M_StartMoveBoxToRoundBelt_ClampB := TRUE; // Method end
END_METHOD

(* This method is used to setting the Fanuc Robot Action " Pickup box from PulloutConveyor , only clampA"
*)
METHOD M_StartPullOutConveyorPickUpBox_ClampA : BOOL
VAR_INPUT
	ClampA_Address : E_PullOutConveyorPosition;
	BoxReady : BOOL; // True : Pullout conveyor box is ready. accroding ClampA target slide is ready or not.
END_VAR
VAR_INST
	_Area : ST_IntToBool;
    _Address_ClampA : ST_IntToBool;
END_VAR
// Set target area is round belt
_Area.nInt := E_RobotArea.PullOutConveyor;
// Select pullout conveyor slide
IF ClampA_Address = E_PullOutConveyorPosition.I3_Slide THEN
	_Address_ClampA.nInt := 1;
ELSIF ClampA_Address = E_PullOutConveyorPosition.I4_Slide THEN
	_Address_ClampA.nInt := 2;
ELSE
	// Wrong command, return
	RETURN ;
END_IF
// Send robot target area data
_DO3.nArea1 := _Area.BitList.Bit0;
_DO3.nArea2 := _Area.BitList.Bit1;
_DO3.nArea3 := _Area.BitList.Bit2;
_DO3.nArea4 := _Area.BitList.Bit3;

// Send robot target address data
_DO3.nAddress1 := _Address_ClampA.BitList.Bit0;
_DO3.nAddress2 := _Address_ClampA.BitList.Bit1;
_DO3.nAddress3 := _Address_ClampA.BitList.Bit2;
_DO3.nAddress4 := _Address_ClampA.BitList.Bit3;
_DO3.nAddress5 := _Address_ClampA.BitList.Bit4;
_DO3.nAddress6 := _Address_ClampA.BitList.Bit5;
_DO3.nAddress7 := _Address_ClampA.BitList.Bit6;

_DO3.bGet := TRUE; // Pickup action
_DO3.bExecute := TRUE;

_DO3.bContinue := BoxReady;

M_StartPullOutConveyorPickUpBox_ClampA := true; // Method end
END_METHOD

(* This method is used to setting the Fanuc Robot Action " Pickup box from PulloutConveyor , only clampB"
*)
METHOD M_StartPullOutConveyorPickUpBox_ClampB : BOOL
VAR_INPUT
	ClampB_Address :E_PullOutConveyorPosition;
	BoxReady : BOOL; // True : Pullout conveyor box is ready. accroding ClampA target slide is ready or not.
END_VAR
VAR_INST
	_Area : ST_IntToBool;
    _Address_ClampB : ST_IntToBool;
END_VAR
// Set target area is round belt
_Area.nInt := E_RobotArea.PullOutConveyor;
// Select pullout conveyor slide
IF ClampB_Address = E_PullOutConveyorPosition.I3_Slide THEN
	_Address_ClampB.nInt := 1;
ELSIF ClampB_Address = E_PullOutConveyorPosition.I4_Slide THEN
	_Address_ClampB.nInt := 2;
ELSE
	// Wrong command, return
	RETURN ;
END_IF

// Send robot target area data
_DO4.nArea1 := _Area.BitList.Bit0;
_DO4.nArea2 := _Area.BitList.Bit1;
_DO4.nArea3 := _Area.BitList.Bit2;
_DO4.nArea4 := _Area.BitList.Bit3;

// Send robot target address data
_DO4.nAddress1 := _Address_ClampB.BitList.Bit0;
_DO4.nAddress2 := _Address_ClampB.BitList.Bit1;
_DO4.nAddress3 := _Address_ClampB.BitList.Bit2;
_DO4.nAddress4 := _Address_ClampB.BitList.Bit3;
_DO4.nAddress5 := _Address_ClampB.BitList.Bit4;
_DO4.nAddress6 := _Address_ClampB.BitList.Bit5;
_DO4.nAddress7 := _Address_ClampB.BitList.Bit6;

_DO4.bGet := TRUE; // Pickup action
_DO4.bExecute := TRUE;

_DO4.bContinue := BoxReady;

M_StartPullOutConveyorPickUpBox_ClampB := true; // Method end
END_METHOD

(* This method is used to setting the Fanuc Robot Action " Pickup box from PulloutConveyor, both clamp"
*)
METHOD M_StartPullOutConveyorPickUpBox_ClampBoth : BOOL
VAR_INPUT
	ClampA_Address : E_PullOutConveyorPosition;
	ClampB_Address : E_PullOutConveyorPosition;
	BoxReady_1 : BOOL; // TRUE : 1st target slide box is ready
	BoxReady_2 : BOOL; // True : 2nd target slide box is ready
END_VAR
VAR_INST
	_Area : ST_IntToBool;
    _Address_ClampA : ST_IntToBool;
    _Address_ClampB : ST_IntToBool;
END_VAR
// Set target area is round belt
_Area.nInt := E_RobotArea.PullOutConveyor;

// Select ClampA target address
IF ClampA_Address = E_PullOutConveyorPosition.I3_Slide THEN
    _Address_ClampA.nInt := 1;
ELSIF ClampA_Address = E_PullOutConveyorPosition.I4_Slide THEN
    _Address_ClampA.nInt := 2;
ELSE
    // Wrong command, return
    RETURN;
END_IF

// Select ClampB target address
IF ClampB_Address = E_PullOutConveyorPosition.I3_Slide THEN
    _Address_ClampB.nInt := 1;
ELSIF ClampB_Address = E_PullOutConveyorPosition.I4_Slide THEN
    _Address_ClampB.nInt := 2;
ELSE
    // Wrong command, return
    RETURN;
END_IF

// Send robot target area data
_DO3.nArea1 := _Area.BitList.Bit0;
_DO3.nArea2 := _Area.BitList.Bit1;
_DO3.nArea3 := _Area.BitList.Bit2;
_DO3.nArea4 := _Area.BitList.Bit3;

_DO4.nArea1 := _Area.BitList.Bit0;
_DO4.nArea2 := _Area.BitList.Bit1;
_DO4.nArea3 := _Area.BitList.Bit2;
_DO4.nArea4 := _Area.BitList.Bit3;

// Send robot target address data
_DO3.nAddress1 := _Address_ClampA.BitList.Bit0;
_DO3.nAddress2 := _Address_ClampA.BitList.Bit1;
_DO3.nAddress3 := _Address_ClampA.BitList.Bit2;
_DO3.nAddress4 := _Address_ClampA.BitList.Bit3;
_DO3.nAddress5 := _Address_ClampA.BitList.Bit4;
_DO3.nAddress6 := _Address_ClampA.BitList.Bit5;
_DO3.nAddress7 := _Address_ClampA.BitList.Bit6;

_DO4.nAddress1 := _Address_ClampB.BitList.Bit0;
_DO4.nAddress2 := _Address_ClampB.BitList.Bit1;
_DO4.nAddress3 := _Address_ClampB.BitList.Bit2;
_DO4.nAddress4 := _Address_ClampB.BitList.Bit3;
_DO4.nAddress5 := _Address_ClampB.BitList.Bit4;
_DO4.nAddress6 := _Address_ClampB.BitList.Bit5;
_DO4.nAddress7 := _Address_ClampB.BitList.Bit6;

_DO3.bGet := TRUE;
_DO4.bGet := TRUE;

_DO3.bExecute := TRUE;
_DO4.bExecute := TRUE;

_DO3.bContinue := BoxReady_1;
_DO4.bContinue := BoxReady_2;

M_StartPullOutConveyorPickUpBox_ClampBoth := true; // Method end
END_METHOD

METHOD PUBLIC M_StartRobotAbsMove : BOOL
VAR_INPUT
	GetBox		: BOOL;
	UseClampA	: BOOL;
	UseClampB   : BOOL;
	Area : E_RobotArea;
	
	
	ClampA_Address	: INT;
	ClampB_Address	: INT;

	BoxReady_1 : BOOL;
	BoxReady_2 : BOOL;
	
END_VAR

VAR_INST
	_Area	: ST_IntToBool;
	_Address_ClampA : ST_IntToBool;
    _Address_ClampB : ST_IntToBool;
END_VAR
//Set target area
_Area.nInt :=Area;

IF UseClampA THEN
	_Address_ClampA.nInt:=ClampA_Address;
	_DO3.nArea1 := _Area.BitList.Bit0;
	_DO3.nArea2 := _Area.BitList.Bit1;
	_DO3.nArea3 := _Area.BitList.Bit2;
	_DO3.nArea4 := _Area.BitList.Bit3;

	_DO3.nAddress1 := _Address_ClampA.BitList.Bit0;
	_DO3.nAddress2 := _Address_ClampA.BitList.Bit1;
	_DO3.nAddress3 := _Address_ClampA.BitList.Bit2;
	_DO3.nAddress4 := _Address_ClampA.BitList.Bit3;
	_DO3.nAddress5 := _Address_ClampA.BitList.Bit4;
	_DO3.nAddress6 := _Address_ClampA.BitList.Bit5;
	_DO3.nAddress7 := _Address_ClampA.BitList.Bit6;
	_DO3.bGet := GetBox;
	_DO3.bExecute := TRUE;
	_DO3.bContinue := BoxReady_1;	
END_IF

IF UseClampB THEN
	_Address_ClampB.nInt:=ClampB_Address;
	_DO4.nArea1 := _Area.BitList.Bit0;
	_DO4.nArea2 := _Area.BitList.Bit1;
	_DO4.nArea3 := _Area.BitList.Bit2;
	_DO4.nArea4 := _Area.BitList.Bit3;
	
	_DO4.nAddress1 := _Address_ClampB.BitList.Bit0;
	_DO4.nAddress2 := _Address_ClampB.BitList.Bit1;
	_DO4.nAddress3 := _Address_ClampB.BitList.Bit2;
	_DO4.nAddress4 := _Address_ClampB.BitList.Bit3;
	_DO4.nAddress5 := _Address_ClampB.BitList.Bit4;
	_DO4.nAddress6 := _Address_ClampB.BitList.Bit5;
	_DO4.nAddress7 := _Address_ClampB.BitList.Bit6;
	_DO4.bGet := GetBox;
	_DO4.bExecute := TRUE;
	_DO4.bContinue := BoxReady_2;	
END_IF

M_StartRobotAbsMove :=TRUE;




















M_StartRobotAbsMove:=TRUE;
END_METHOD

METHOD M_StartWarehouseMoveAction_ClampA : BOOL
VAR_INPUT
	WareHouseSelect : E_WareHouse;
	Info : ST_WareHouseCoordinates; // Input Warehouse with robot move parameter for pickup box;
	ClampAction :E_ClampAction;
	BoxReady : BOOL;
END_VAR
VAR_OUTPUT
	Error : BOOL;
	ErrMsg :T_MaxString;
END_VAR
VAR_INST
	_Layer : ST_IntToBool;
	_Slide : ST_IntToBool;
END_VAR
// Set target warehouse
CASE WareHouseSelect OF
    E_WareHouse.WareHouseA:
        _DO1.bTargetWareHouseA := TRUE;
        _DO1.bTargetWareHouseB := FALSE;
    E_WareHouse.WareHouseB:
        _DO1.bTargetWareHouseA := FALSE;
        _DO1.bTargetWareHouseB := TRUE;
ELSE
    _DO1.bTargetWareHouseA := FALSE;
    _DO1.bTargetWareHouseB := FALSE;
    Error                  := TRUE;
    ErrMsg                 := 'ClampA target warehouse out of range';
	RETURN;
END_CASE

// Set Warehouse coordinates
_Layer.nInt := info.Layer;
_Slide.nInt := info.Slide;

// Send Layer data to robot
_DO1.nLayer1 := _Layer.BitList.Bit0;
_DO1.nLayer2 := _Layer.BitList.Bit1;
_DO1.nLayer3 := _Layer.BitList.Bit2;
_DO1.nLayer4 := _Layer.BitList.Bit3;

// Send Slide data to Robot
_DO1.nSlide1 := _Slide.BitList.Bit0;
_DO1.nSlide2 := _Slide.BitList.Bit1;
_DO1.nSlide3 := _Slide.BitList.Bit2;
_DO1.nSlide4 := _Slide.BitList.Bit3;
_DO1.nSlide5 := _Slide.BitList.Bit4;

// Send clamp action to robot
CASE ClampAction OF
	E_ClampAction.PickUp:
		_DO1.bGet := TRUE;
	E_ClampAction.Place:
		_DO1.bGet := FALSE;
ELSE
	Error := TRUE;
	ErrMsg := 'Clamp action not defined';
	RETURN;
END_CASE

// Send action data to robot
_DO1.bExecute := NOT Error;
_DO1.bContinue := BoxReady;
M_StartWarehouseMoveAction_ClampA := NOT Error; // Method end
END_METHOD

METHOD M_StartWarehouseMoveAction_ClampB : BOOL
VAR_INPUT
	WareHouseSelect : E_WareHouse;
	Info : ST_WareHouseCoordinates; // Input Warehouse with robot move parameter for pickup box;
	ClampAction :E_ClampAction;
	BoxReady : BOOL;
END_VAR
VAR_OUTPUT
	Error : BOOL;
	ErrMsg :T_MaxString;
END_VAR
VAR_INST
	_Layer : ST_IntToBool;
	_Slide : ST_IntToBool;
END_VAR
// Set target warehouse
CASE WareHouseSelect OF
    E_WareHouse.WareHouseA:
        _DO2.bTargetWareHouseA := TRUE;
        _DO2.bTargetWareHouseB := FALSE;
    E_WareHouse.WareHouseB:
        _DO2.bTargetWareHouseA := FALSE;
        _DO2.bTargetWareHouseB := TRUE;
ELSE
    _DO2.bTargetWareHouseA := FALSE;
    _DO2.bTargetWareHouseB := FALSE;
    Error                  := TRUE;
    ErrMsg                 := 'ClampB target warehouse out of range';
	RETURN;
END_CASE

// Set Warehouse coordinates
_Layer.nInt := info.Layer;
_Slide.nInt := info.Slide;

// Send Layer data to robot
_DO2.nLayer1 := _Layer.BitList.Bit0;
_DO2.nLayer2 := _Layer.BitList.Bit1;
_DO2.nLayer3 := _Layer.BitList.Bit2;
_DO2.nLayer4 := _Layer.BitList.Bit3;

// Send Slide data to Robot
_DO2.nSlide1 := _Slide.BitList.Bit0;
_DO2.nSlide2 := _Slide.BitList.Bit1;
_DO2.nSlide3 := _Slide.BitList.Bit2;
_DO2.nSlide4 := _Slide.BitList.Bit3;
_DO2.nSlide5 := _Slide.BitList.Bit4;

// Send clamp action to robot
CASE ClampAction OF
	E_ClampAction.PickUp:
		_DO2.bGet := TRUE;
	E_ClampAction.Place:
		_DO2.bGet := FALSE;
ELSE
	Error := TRUE;
	ErrMsg := 'Clamp action not defined';
	RETURN;
END_CASE

// Send action data to robot
_DO2.bExecute := NOT Error;
_DO2.bContinue := BoxReady;

M_StartWarehouseMoveAction_ClampB := NOT Error; // Method End
END_METHOD

METHOD M_StartWarehouseMoveAction_ClampBoth : BOOL
VAR_INPUT
	WareHouseSelect : E_WareHouse;
	ClampA_Info : ST_WareHouseCoordinates; // Input Warehouse with robot move parameter for pickup box;
	ClampB_Info : ST_WareHouseCoordinates; // Input Warehouse with robot move parameter for pickup box;
	ClampAction_A : E_ClampAction;
	ClampAction_B : E_ClampAction;
	BoxReady_1st : BOOL; // Box is arrived, ready to pickup
	BoxReady_2nd : BOOL; // Box is arrived, ready to pickup
END_VAR
VAR_OUTPUT
	Error : BOOL;
	ErrMsg :T_MaxString;
END_VAR
VAR_INST
	_LayerClampA :ST_IntToBool;
	_SlideClampA : ST_IntToBool;
	_LayerClampB : ST_IntToBool;
	_SLideClampB : ST_IntToBool;
END_VAR
// Set target warehouse
CASE WareHouseSelect OF
    E_WareHouse.WareHouseA:
        _DO1.bTargetWareHouseA := TRUE;
        _DO1.bTargetWareHouseB := FALSE;
        _DO2.bTargetWareHouseA := TRUE;
        _DO2.bTargetWareHouseB := FALSE;
    E_WareHouse.WareHouseB:
        _DO1.bTargetWareHouseA := FALSE;
        _DO1.bTargetWareHouseB := TRUE;
        _DO2.bTargetWareHouseA := FALSE;
        _DO2.bTargetWareHouseB := TRUE;
ELSE
    _DO1.bTargetWareHouseA := FALSE;
    _DO1.bTargetWareHouseB := FALSE;
    _DO2.bTargetWareHouseA := FALSE;
    _DO2.bTargetWareHouseB := FALSE;
    Error                  := TRUE;
    ErrMsg                 := 'Clamp target warehouse out of range';
    RETURN;
END_CASE

// Assign coordinates 
_LayerClampA.nInt := ClampA_Info.Layer;
_SlideClampA.nInt := ClampA_Info.Slide;
_LayerClampB.nInt := ClampB_Info.Layer;
_SlideClampB.nInt := ClampB_Info.Slide;

// Send Layer data to Robot
_DO1.nLayer1 := _LayerClampA.BitList.Bit0;
_DO1.nLayer2 := _LayerClampA.BitList.Bit1;
_DO1.nLayer3 := _LayerClampA.BitList.Bit2;
_DO1.nLayer4 := _LayerClampA.BitList.Bit3;
_DO2.nLayer1 := _LayerClampB.BitList.Bit0;
_DO2.nLayer2 := _LayerClampB.BitList.Bit1;
_DO2.nLayer3 := _LayerClampB.BitList.Bit2;
_DO2.nLayer4 := _LayerClampB.BitList.Bit3;
// Send Slide data to Robot
_DO1.nSlide1 := _SlideClampA.BitList.Bit0;
_DO1.nSlide2 := _SlideClampA.BitList.Bit1;
_DO1.nSlide3 := _SlideClampA.BitList.Bit2;
_DO1.nSlide4 := _SlideClampA.BitList.Bit3;
_DO1.nSlide5 := _SlideClampA.BitList.Bit4;

_DO2.nSlide1 := _SlideClampB.BitList.Bit0;
_DO2.nSlide2 := _SlideClampB.BitList.Bit1;
_DO2.nSlide3 := _SlideClampB.BitList.Bit2;
_DO2.nSlide4 := _SlideClampB.BitList.Bit3;
_DO2.nSlide5 := _SlideClampB.BitList.Bit4;

// Set clamp action 
CASE ClampAction_A OF
	E_ClampAction.PickUp:
		_DO1.bGet := TRUE;
	E_ClampAction.Place:
		_DO1.bGet := FALSE;
ELSE
	Error := TRUE;
	ErrMsg := 'ClampA action not defined';
	RETURN;
END_CASE

// Set clamp action
CASE ClampAction_B OF
	E_ClampAction.PickUp:
		_DO2.bGet := TRUE;
	E_ClampAction.Place:
		_DO2.bGet := FALSE;
ELSE
	Error := TRUE;
	ErrMsg := 'ClampB action not defined';
	RETURN;	
END_CASE

// set execute
_DO1.bExecute := NOT Error;
_DO2.bExecute := NOT Error;

_DO1.bContinue := BoxReady_1st;
_DO2.bContinue := BoxReady_2nd;

M_StartWarehouseMoveAction_ClampBoth := NOT Error; // Method end
END_METHOD

METHOD M_StartWareHousePickUpBox_ClampA : Bool
VAR_INPUT
	WareHouseSelect : E_WareHouse;
	Info : ST_WareHouseCoordinates; // Input Warehouse with robot move parameter for pickup box;
	BoxReady_1st : BOOL;
END_VAR
VAR_INST
	_Layer : ST_IntToBool;
	_Slide : ST_IntToBool;
END_VAR
// Send target warehouse to robot
IF WareHouseSelect = E_WareHouse.WareHouseA THEN
	_DO1.bTargetWareHouseA := TRUE;
	_DO1.bTargetWareHouseB := FALSE;
ELSIF WareHouseSelect = E_WareHouse.WareHouseB THEN
	_DO1.bTargetWareHouseA := FALSE;
	_DO1.bTargetWareHouseB := TRUE;
ELSE
	_DO1.bTargetWareHouseA := FALSE;
	_DO1.bTargetWareHouseB := FALSE;
END_IF

// Assign coordinates 
_Layer.nInt := info.Layer;
_Slide.nInt := info.Slide;

// Send Layer data to Robot
_DO1.nLayer1 := _Layer.BitList.Bit0;
_DO1.nLayer2 := _Layer.BitList.Bit1;
_DO1.nLayer3 := _Layer.BitList.Bit2;
_DO1.nLayer4 := _Layer.BitList.Bit3;

// Send Slide data to Robot
_DO1.nSlide1 := _Slide.BitList.Bit0;
_DO1.nSlide2 := _Slide.BitList.Bit1;
_DO1.nSlide3 := _Slide.BitList.Bit2;
_DO1.nSlide4 := _Slide.BitList.Bit3;
_DO1.nSlide5 := _Slide.BitList.Bit4;

// Send action data to robot
_DO1.bGet := TRUE; // PickUp
// Send execute command 
_DO1.bExecute := TRUE;
_DO1.bContinue := BoxReady_1st;
M_StartWareHousePickUpBox_ClampA := TRUE; // Method end
END_METHOD

METHOD M_StartWareHousePickUpBox_ClampB : BOOL
VAR_INPUT
	WareHouseSelect : E_WareHouse;
	Info : ST_WareHouseCoordinates; // Input Warehouse with robot move parameter for pickup box;
	BoxReady_2nd : BOOL;
END_VAR
VAR_INST
	_Layer : ST_IntToBool;
	_Slide : ST_IntToBool;
END_VAR
// Send target warehouse to robot
IF WareHouseSelect = E_WareHouse.WareHouseA THEN
    _DO2.bTargetWareHouseA := TRUE;
    _DO2.bTargetWareHouseB := FALSE;
ELSIF WareHouseSelect = E_WareHouse.WareHouseB THEN
    _DO2.bTargetWareHouseA := FALSE;
    _DO2.bTargetWareHouseB := TRUE;
ELSE
    _DO2.bTargetWareHouseA := FALSE;
    _DO2.bTargetWareHouseB := FALSE;
END_IF

// Assign coordinates 
_Layer.nInt := info.Layer;
_Slide.nInt := info.Slide;

// Send Layer data to Robot
_DO2.nLayer1 := _Layer.BitList.Bit0;
_DO2.nLayer2 := _Layer.BitList.Bit1;
_DO2.nLayer3 := _Layer.BitList.Bit2;
_DO2.nLayer4 := _Layer.BitList.Bit3;

// Send Slide data to Robot
_DO2.nSlide1 := _Slide.BitList.Bit0;
_DO2.nSlide2 := _Slide.BitList.Bit1;
_DO2.nSlide3 := _Slide.BitList.Bit2;
_DO2.nSlide4 := _Slide.BitList.Bit3;
_DO2.nSlide5 := _Slide.BitList.Bit4;

// Send action data to robot
_DO2.bGet := TRUE; // PickUp
// Send execute command 
_DO2.bExecute := TRUE;
_DO2.bContinue:=BoxReady_2nd;
M_StartWareHousePickUpBox_ClampB := TRUE; // Method end
END_METHOD

METHOD M_StartWareHousePickUpBox_ClampBoth : BOOL
VAR_INPUT
	WareHouseSelect : E_WareHouse;
	ClampA_Info : ST_WareHouseCoordinates; // Input Warehouse with robot move parameter for pickup box;
	ClampB_Info : ST_WareHouseCoordinates; // Input Warehouse with robot move parameter for pickup box;
	BoxReady_1st : BOOL; // Box is arrived, ready to pickup
	BoxReady_2nd : BOOL; // Box is arrived, ready to pickup
END_VAR
VAR_OUTPUT
	Error : BOOL;
	ErrMsg :T_MaxString;
END_VAR
VAR_INST
	_LayerClampA : ST_IntToBool;
	_SlideClampA : ST_IntToBool;
	_LayerClampB : ST_IntToBool;
	_SlideClampB : ST_IntToBool;
END_VAR
// Set target warehouse
CASE WareHouseSelect OF
    E_WareHouse.WareHouseA:
        _DO1.bTargetWareHouseA := TRUE;
        _DO1.bTargetWareHouseB := FALSE;
        _DO2.bTargetWareHouseA := TRUE;
        _DO2.bTargetWareHouseB := FALSE;
    E_WareHouse.WareHouseB:
        _DO1.bTargetWareHouseA := FALSE;
        _DO1.bTargetWareHouseB := TRUE;
        _DO2.bTargetWareHouseA := FALSE;
        _DO2.bTargetWareHouseB := TRUE;
ELSE
    _DO1.bTargetWareHouseA := FALSE;
    _DO1.bTargetWareHouseB := FALSE;
    _DO2.bTargetWareHouseA := FALSE;
    _DO2.bTargetWareHouseB := FALSE;
    Error                  := TRUE;
    ErrMsg                 := 'Clamp target warehouse out of range';
    RETURN;
END_CASE

// Assign coordinates 
_LayerClampA.nInt := ClampA_Info.Layer;
_SlideClampA.nInt := ClampA_Info.Slide;
_LayerClampB.nInt := ClampB_Info.Layer;
_SlideClampB.nInt := ClampB_Info.Slide;

// Send Layer data to Robot
_DO1.nLayer1 := _LayerClampA.BitList.Bit0;
_DO1.nLayer2 := _LayerClampA.BitList.Bit1;
_DO1.nLayer3 := _LayerClampA.BitList.Bit2;
_DO1.nLayer4 := _LayerClampA.BitList.Bit3;

_DO2.nLayer1 := _LayerClampB.BitList.Bit0;
_DO2.nLayer2 := _LayerClampB.BitList.Bit1;
_DO2.nLayer3 := _LayerClampB.BitList.Bit2;
_DO2.nLayer4 := _LayerClampB.BitList.Bit3;
// Send Slide data to Robot
_DO1.nSlide1 := _SlideClampA.BitList.Bit0;
_DO1.nSlide2 := _SlideClampA.BitList.Bit1;
_DO1.nSlide3 := _SlideClampA.BitList.Bit2;
_DO1.nSlide4 := _SlideClampA.BitList.Bit3;
_DO1.nSlide5 := _SlideClampA.BitList.Bit4;

_DO2.nSlide1 := _SlideClampB.BitList.Bit0;
_DO2.nSlide2 := _SlideClampB.BitList.Bit1;
_DO2.nSlide3 := _SlideClampB.BitList.Bit2;
_DO2.nSlide4 := _SlideClampB.BitList.Bit3;
_DO2.nSlide5 := _SlideClampB.BitList.Bit4;

// Send action data to robot
_DO1.bGet := TRUE; // ClampA PickUp
_DO2.bGet := TRUE; // ClampB PickUp
// Send execute command 
_DO1.bExecute := NOT Error;
_DO2.bExecute := NOT Error;

_DO1.bContinue := BoxReady_1st;
_DO2.bContinue := BoxReady_2nd;

M_StartWareHousePickUpBox_ClampBoth := NOT Error; // Method end
END_METHOD

METHOD M_StartWareHousePlaceBox_ClampA : Bool
VAR_INPUT
	WareHouseSelect : E_WareHouse;
	Info : ST_WareHouseCoordinates; // Input Warehouse with robot move parameter for pickup box;
	BoxReady_1st : BOOL;
END_VAR
VAR_INST
	_Layer : ST_IntToBool;
	_Slide : ST_IntToBool;
END_VAR
// Send target warehouse to robot
IF WareHouseSelect = E_WareHouse.WareHouseA THEN
	_DO1.bTargetWareHouseA := TRUE;
	_DO1.bTargetWareHouseB := FALSE;
ELSIF WareHouseSelect = E_WareHouse.WareHouseB THEN
	_DO1.bTargetWareHouseA := FALSE;
	_DO1.bTargetWareHouseB := TRUE;
ELSE
	_DO1.bTargetWareHouseA := FALSE;
	_DO1.bTargetWareHouseB := FALSE;
END_IF

// Assign coordinates 
_Layer.nInt := info.Layer;
_Slide.nInt := info.Slide;

// Send Layer data to Robot
_DO1.nLayer1 := _Layer.BitList.Bit0;
_DO1.nLayer2 := _Layer.BitList.Bit1;
_DO1.nLayer3 := _Layer.BitList.Bit2;
_DO1.nLayer4 := _Layer.BitList.Bit3;

// Send Slide data to Robot
_DO1.nSlide1 := _Slide.BitList.Bit0;
_DO1.nSlide2 := _Slide.BitList.Bit1;
_DO1.nSlide3 := _Slide.BitList.Bit2;
_DO1.nSlide4 := _Slide.BitList.Bit3;
_DO1.nSlide5 := _Slide.BitList.Bit4;

// Send action data to robot
_DO1.bGet := FALSE; // PickUp
// Send execute command 
_DO1.bExecute := TRUE;
_DO1.bContinue := BoxReady_1st;
M_StartWareHousePlaceBox_ClampA := TRUE; // Method end
END_METHOD

METHOD M_StartWareHousePlaceBox_ClampB : BOOL
VAR_INPUT
	WareHouseSelect : E_WareHouse;
	Info : ST_WareHouseCoordinates; // Input Warehouse with robot move parameter for pickup box;
	BoxReady_2nd : BOOL;
END_VAR
VAR_INST
	_Layer : ST_IntToBool;
	_Slide : ST_IntToBool;
END_VAR
// Send target warehouse to robot
IF WareHouseSelect = E_WareHouse.WareHouseA THEN
    _DO2.bTargetWareHouseA := TRUE;
    _DO2.bTargetWareHouseB := FALSE;
ELSIF WareHouseSelect = E_WareHouse.WareHouseB THEN
    _DO2.bTargetWareHouseA := FALSE;
    _DO2.bTargetWareHouseB := TRUE;
ELSE
    _DO2.bTargetWareHouseA := FALSE;
    _DO2.bTargetWareHouseB := FALSE;
END_IF

// Assign coordinates 
_Layer.nInt := info.Layer;
_Slide.nInt := info.Slide;

// Send Layer data to Robot
_DO2.nLayer1 := _Layer.BitList.Bit0;
_DO2.nLayer2 := _Layer.BitList.Bit1;
_DO2.nLayer3 := _Layer.BitList.Bit2;
_DO2.nLayer4 := _Layer.BitList.Bit3;

// Send Slide data to Robot
_DO2.nSlide1 := _Slide.BitList.Bit0;
_DO2.nSlide2 := _Slide.BitList.Bit1;
_DO2.nSlide3 := _Slide.BitList.Bit2;
_DO2.nSlide4 := _Slide.BitList.Bit3;
_DO2.nSlide5 := _Slide.BitList.Bit4;

// Send action data to robot
_DO2.bGet := FALSE; // PickUp
// Send execute command 
_DO2.bExecute := TRUE;
_DO2.bContinue:=BoxReady_2nd;
M_StartWareHousePlaceBox_ClampB := TRUE; // Method end
END_METHOD

METHOD M_StartWareHousePlaceUpBox_ClampBoth : BOOL
VAR_INPUT
	WareHouseSelect : E_WareHouse;
	ClampA_Info : ST_WareHouseCoordinates; // Input Warehouse with robot move parameter for pickup box;
	ClampB_Info : ST_WareHouseCoordinates; // Input Warehouse with robot move parameter for pickup box;
	BoxReady_1st : BOOL; // Box is arrived, ready to pickup
	BoxReady_2nd : BOOL; // Box is arrived, ready to pickup
END_VAR
VAR_OUTPUT
	Error : BOOL;
	ErrMsg :T_MaxString;
END_VAR
VAR_INST
	_LayerClampA : ST_IntToBool;
	_SlideClampA : ST_IntToBool;
	_LayerClampB : ST_IntToBool;
	_SlideClampB : ST_IntToBool;
END_VAR
// Set target warehouse
CASE WareHouseSelect OF
    E_WareHouse.WareHouseA:
        _DO1.bTargetWareHouseA := TRUE;
        _DO1.bTargetWareHouseB := FALSE;
        _DO2.bTargetWareHouseA := TRUE;
        _DO2.bTargetWareHouseB := FALSE;
    E_WareHouse.WareHouseB:
        _DO1.bTargetWareHouseA := FALSE;
        _DO1.bTargetWareHouseB := TRUE;
        _DO2.bTargetWareHouseA := FALSE;
        _DO2.bTargetWareHouseB := TRUE;
ELSE
    _DO1.bTargetWareHouseA := FALSE;
    _DO1.bTargetWareHouseB := FALSE;
    _DO2.bTargetWareHouseA := FALSE;
    _DO2.bTargetWareHouseB := FALSE;
    Error                  := TRUE;
    ErrMsg                 := 'Clamp target warehouse out of range';
    RETURN;
END_CASE

// Assign coordinates 
_LayerClampA.nInt := ClampA_Info.Layer;
_SlideClampA.nInt := ClampA_Info.Slide;
_LayerClampB.nInt := ClampB_Info.Layer;
_SlideClampB.nInt := ClampB_Info.Slide;

// Send Layer data to Robot
_DO1.nLayer1 := _LayerClampA.BitList.Bit0;
_DO1.nLayer2 := _LayerClampA.BitList.Bit1;
_DO1.nLayer3 := _LayerClampA.BitList.Bit2;
_DO1.nLayer4 := _LayerClampA.BitList.Bit3;

_DO2.nLayer1 := _LayerClampB.BitList.Bit0;
_DO2.nLayer2 := _LayerClampB.BitList.Bit1;
_DO2.nLayer3 := _LayerClampB.BitList.Bit2;
_DO2.nLayer4 := _LayerClampB.BitList.Bit3;
// Send Slide data to Robot
_DO1.nSlide1 := _SlideClampA.BitList.Bit0;
_DO1.nSlide2 := _SlideClampA.BitList.Bit1;
_DO1.nSlide3 := _SlideClampA.BitList.Bit2;
_DO1.nSlide4 := _SlideClampA.BitList.Bit3;
_DO1.nSlide5 := _SlideClampA.BitList.Bit4;

_DO2.nSlide1 := _SlideClampB.BitList.Bit0;
_DO2.nSlide2 := _SlideClampB.BitList.Bit1;
_DO2.nSlide3 := _SlideClampB.BitList.Bit2;
_DO2.nSlide4 := _SlideClampB.BitList.Bit3;
_DO2.nSlide5 := _SlideClampB.BitList.Bit4;

// Send action data to robot
_DO1.bGet := FALSE; // ClampA PickUp
_DO2.bGet := FALSE; // ClampB PickUp
// Send execute command 
_DO1.bExecute := NOT Error;
_DO2.bExecute := NOT Error;

_DO1.bContinue := BoxReady_1st;
_DO2.bContinue := BoxReady_2nd;

M_StartWareHousePlaceUpBox_ClampBoth := NOT Error; // Method end
END_METHOD

METHOD M_SwitchRSR3 : BOOL
VAR_INPUT
END_VAR
END_METHOD

PROPERTY Read_OffsetP : INT
GET
Read_OffsetP := _DI6;
END_GET
END_PROPERTY

PROPERTY Read_OffsetR : INT
GET
Read_OffsetR := _DI7;
END_GET
END_PROPERTY

PROPERTY Read_OffsetW : INT
GET
Read_OffsetW := _DI5;
END_GET
END_PROPERTY

PROPERTY Read_OffsetX : INT
GET
Read_OffsetX := _DI2;
END_GET
END_PROPERTY

PROPERTY Read_OffsetY : INT
GET
Read_OffsetY := _DI3;
END_GET
END_PROPERTY

PROPERTY Read_OffsetZ : INT
GET
Read_OffsetZ := _DI4;
END_GET
END_PROPERTY

PROPERTY ReadDataCommand : BOOL;
SET
_DO6.ReadPara_Execute := BOOL_TO_BIT(ReadDataCommand);
END_SET
END_PROPERTY

PROPERTY ReadWrite_Address : Int
SET
_Do14 := ReadWrite_Address;
END_SET
END_PROPERTY

PROPERTY ReadWrite_Area : E_RobotArea
SET
_Do13 := ReadWrite_Area;
END_SET
END_PROPERTY

(* This variable is used to define read/write offset data clamp A
*)
PROPERTY ReadWrite_ClampA : BOOL
SET
_DO6.ClampA :=  BOOL_TO_BIT(ReadWrite_ClampA );
END_SET
END_PROPERTY

(* This variable is used to define read/write offset data clamp B
*)
PROPERTY ReadWrite_ClampB : BOOL
SET
_DO6.ClampB :=BOOL_TO_BIT( ReadWrite_ClampB);
END_SET
END_PROPERTY

(* This variable is used to define read/write offset data warehouse A
*)
PROPERTY ReadWrite_WareHouseA : BOOL
SET
_DO6.WareHouseA := BOOL_TO_BIT(ReadWrite_WareHouseA);
END_SET
END_PROPERTY

(* This variable is used to define read/write offset data warehouse B
*)
PROPERTY ReadWrite_WareHouseB : BOOL
SET
_DO6.WarehouseB := BOOL_TO_BIT(ReadWrite_WareHouseB);
END_SET
END_PROPERTY

(*Fanuc robot ready to work for command (Warehouse、AbsMove)*)
PROPERTY ReadyOperation : Bool
GET
ReadyOperation := _RSR1_Ready;
END_GET
END_PROPERTY

PROPERTY ReadySetParameter : Bool
GET
ReadySetParameter := _RSR3_Ready;
END_GET
END_PROPERTY

METHOD ReBoot
VAR_INPUT
END_VAR
eState := E_MethodStatus_Basic.STATE_DORMANT;
END_METHOD

PROPERTY SlideIndex : INT
SET
_DO16 := SlideIndex;
END_SET
END_PROPERTY

PROPERTY Status : ST_FanucUI1
GET
Status := _UI1;
END_GET
END_PROPERTY

METHOD Update : BOOL
VAR_INPUT
END_VAR
// Robot -> PLC 4 byte 外圍設備Output(Fanuc Robot的外圍)
MEMMOVE(
destAddr:=ADR(_UO1)
,srcAddr:=ADR(_rawIn_UI[0])
,n:=4
);

// PLC -> Robot 外圍設備Input(Fanuc Robot的外圍)
MEMMOVE(
destAddr:=ADR(_rawOut_UO[0])
,srcAddr:=ADR(_UI1)
,n:=4
);
// PLC -> Robot Digital Output 2byte(send the command to Fanuc Robot), Warehouse Robot move ClampA
MEMMOVE(
destAddr:=ADR(_rawOut_DO[0])
,srcAddr:=ADR(_DO1)
,n:=2 
);
// PLC -> Robot Digital Output 2byte(send the command to Fanuc Robot), Warehouse Robot move ClampB
MEMMOVE(
destAddr:=ADR(_rawOut_DO[2])
,srcAddr:=ADR(_DO2)
,n:=2 
);
// PLC -> Robot Digital Output 2byte(send the command to Fanuc Robot), ABS Robot move ClampA
MEMMOVE(
destAddr:=ADR(_rawOut_DO[4])
,srcAddr:=ADR(_DO3)
,n:=2 
);
// PLC -> Robot Digital Output 2byte(send the command to Fanuc Robot), ABS Robot move ClampA
MEMMOVE(
destAddr:=ADR(_rawOut_DO[6])
,srcAddr:=ADR(_DO4)
,n:=2 
);
// PLC -> Robot Digital output 2byte(send the command to Fanuc Robot), General Command
MEMMOVE(
destAddr:=ADR(_rawOut_DO[8])
,srcAddr:=ADR(_DO5)
,n:=2 
);
MEMMOVE(
destAddr:=ADR(_rawOut_DO[10])
,srcAddr:=ADR(_DO6)
,n:=2 
);
MEMMOVE(
destAddr:=ADR(_rawOut_DO[12])
,srcAddr:=ADR(_DO7)
,n:=2 
);
MEMMOVE(
destAddr:=ADR(_rawOut_DO[14])
,srcAddr:=ADR(_DO8)
,n:=2 
);
MEMMOVE(
destAddr:=ADR(_rawOut_DO[16])
,srcAddr:=ADR(_DO9)
,n:=2 
);

MEMMOVE(
destAddr:=ADR(_rawOut_DO[18])
,srcAddr:=ADR(_DO10)
,n:=2 
);
MEMMOVE(
destAddr:=ADR(_rawOut_DO[20])
,srcAddr:=ADR(_DO11)
,n:=2 
);
MEMMOVE(
destAddr:=ADR(_rawOut_DO[22])
,srcAddr:=ADR(_DO12)
,n:=2 
);
MEMMOVE(
destAddr:=ADR(_rawOut_DO[24])
,srcAddr:=ADR(_DO13)
,n:=2 
);
MEMMOVE(
destAddr:=ADR(_rawOut_DO[26])
,srcAddr:=ADR(_DO14)
,n:=2 
);
MEMMOVE(
destAddr:=ADR(_rawOut_DO[28])
,srcAddr:=ADR(_DO15)
,n:=2 
);
MEMMOVE(
destAddr:=ADR(_rawOut_DO[30])
,srcAddr:=ADR(_DO16)
,n:=2 
);


// Robot -> PLC Digital Input 3byte(Send Robot Status to PLC), All service
MEMMOVE(
destAddr:=ADR(_DI1)
,srcAddr:=ADR(_rawIn_DI[0])
,n:=3
);

MEMMOVE(
destAddr:=ADR(_DI2)
,srcAddr:=ADR(_rawIn_DI[3])
,n:=2
);
MEMMOVE(
destAddr:=ADR(_DI3)
,srcAddr:=ADR(_rawIn_DI[5])
,n:=2
);
MEMMOVE(
destAddr:=ADR(_DI4)
,srcAddr:=ADR(_rawIn_DI[7])
,n:=2
);
MEMMOVE(
destAddr:=ADR(_DI5)
,srcAddr:=ADR(_rawIn_DI[9])
,n:=2
);
MEMMOVE(
destAddr:=ADR(_DI6)
,srcAddr:=ADR(_rawIn_DI[11])
,n:=2
);
MEMMOVE(
destAddr:=ADR(_DI7)
,srcAddr:=ADR(_rawIn_DI[13])
,n:=2
);
MEMMOVE(
destAddr:=ADR(_DI8)
,srcAddr:=ADR(_rawIn_DI[15])
,n:=2
);
MEMMOVE(
destAddr:=ADR(_DI9)
,srcAddr:=ADR(_rawIn_DI[17])
,n:=2
);
MEMMOVE(
destAddr:=ADR(_DI10)
,srcAddr:=ADR(_rawIn_DI[19])
,n:=2
);
MEMMOVE(
destAddr:=ADR(_DI11)
,srcAddr:=ADR(_rawIn_DI[21])
,n:=2
);
MEMMOVE(
destAddr:=ADR(_DI12)
,srcAddr:=ADR(_rawIn_DI[23])
,n:=2
);

// Robot Status com
qEnable:=_UO1.UO01_CmdEnabled AND _UO1.UO02_SystemReady;
Error:=Fault();

// Velocity Command transfer
_DO5.VelocityBit0 := _VelocityCommand.BitList.Bit0;
_DO5.VelocityBit1 := _VelocityCommand.BitList.Bit1;
_DO5.VelocityBit2 := _VelocityCommand.BitList.Bit2;
_DO5.VelocityBit3 := _VelocityCommand.BitList.Bit3;
_DO5.VelocityBit4 := _VelocityCommand.BitList.Bit4;
_DO5.VelocityBit5 := _VelocityCommand.BitList.Bit5;
_DO5.VelocityBit6 := _VelocityCommand.BitList.Bit6;
_DO5.VelocityBit7 := _VelocityCommand.BitList.Bit7;
END_METHOD

{attribute 'monitoring' := 'variable'}
PROPERTY VelocityCommand : Int
GET
VelocityCommand :=_VelocityCommand.nInt;
END_GET
SET
_VelocityCommand.nInt :=VelocityCommand;
END_SET
END_PROPERTY

PROPERTY WareHouseClampA_Handshake : ST_Fanuc_WarehouseHandshake
GET
WareHouseClampA_Handshake := _DO1;
END_GET
SET
// Outside -> FB 
_DO1 := WareHouseClampA_Handshake;
END_SET
END_PROPERTY

PROPERTY WareHouseClampB_Handshake : ST_Fanuc_WarehouseHandshake
GET
WareHouseClampB_Handshake := _DO2;
END_GET
SET
// Outside -> FB 
_DO2 := WareHouseClampB_Handshake;
END_SET
END_PROPERTY

PROPERTY Write_OffsetP : INT
SET
_DI11 := Write_OffsetP;
END_SET
END_PROPERTY

PROPERTY Write_OffsetR : INT
SET
_DO12 := Write_OffsetR;
END_SET
END_PROPERTY

PROPERTY Write_OffsetW : INT
SET
_DO10 := Write_OffsetW;
END_SET
END_PROPERTY

PROPERTY Write_OffsetX : INT
SET
_DO7 := Write_OffsetX;
END_SET
END_PROPERTY

PROPERTY Write_OffsetY : INT
SET
_DO8 := Write_OffsetY;
END_SET
END_PROPERTY

PROPERTY Write_OffsetZ : INT
SET
_DO9 := Write_OffsetZ;
END_SET
END_PROPERTY

PROPERTY WriteDataCommand : bool;
SET
_DO6.WritePara_Execute := WriteDataCommand;
END_SET
END_PROPERTY

END_FUNCTION_BLOCK

// ---- Library/20_MachineUnits/21_StorageArea/Service/FB_FeedInEmptyBoxWithRobot.TcPOU
FUNCTION_BLOCK FB_FeedInEmptyBoxWithRobot EXTENDS FB_ObjectBase_V2 IMPLEMENTS IBasicElement
VAR_INPUT
    // Below are the components being controlled.
    Robot           : REFERENCE TO FB_FanucRobot_Basic; // Fanuc Robot
    PullOutConveyor : REFERENCE TO FB_PullOutConveyorAction; // Allocated area pull out conveyor
    DiffSizeCV  : REFERENCE TO FB_Motor; // Allocated area feed in conveyor(diff and same size conveyor)
	SameSizeCV : REFERENCE TO FB_Motor;
    WareHouse       : REFERENCE TO FB_WareHouse; // Storage area warehouse A and warehouse B conveyor and sensor
    //SameSizeFullSensor : REFERENCE TO BOOL; 				 // Because the same size sensor implement FB_ConveyorSameSize, so use reference to connect it
    Info  : ST_FeedInEmptyBox_Info; // Setting the feedin emptybox action's parameter
    Input : REFERENCE TO ST_InputTable;
    Stop  : BOOL;
END_VAR
VAR_OUTPUT
END_VAR
VAR
    tonPlaceSensorDelay    : TON;
    tonFeedInConveyorDelay : TON;
    tonTimeOut             : TON;
    tonFeedBoxTimeout      : TON;
    strStatus              : STRING;
    _UniqueErrorCode       : STRING;
    _Abort                 : BOOL;
    uiResumeStep           : DINT;
    PreviousStrStatus      : STRING;
    PreviousErrorCode      : STRING;
END_VAR

SUPER^.A10_StateControl();
tonPlaceSensorDelay(PT:=T#1S);
tonFeedInConveyorDelay(PT:=T#500MS);

ACTION A00_BasicUnits:
tonTimeOut(PT:=T#60S);
tonFeedBoxTimeout(PT:=T#15s);
END_ACTION

METHOD M_CheckCommand : BOOL
VAR_INPUT
END_VAR

VAR_INST
	CheckBehavior : BOOL; // True : Behavior is correct
	CheckWareHouseSetting : BOOL; // True : WareHouse setting is correct
	CheckPullOutConveyorSetting : BOOL; // True : PullOut Conveyor setting is correct
	CheckPickUpArea : BOOL; // True : PickUp Area is correct
	CheckPlaceArea : BOOL; // True : Place Area is correct
END_VAR
// Memory clear
CheckBehavior := FALSE;
// Check command is correct
IF info.ClampA_Setting.Behavior = E_ClampWork.Work OR info.ClampB_Setting.Behavior = E_ClampWork.Work THEN
	CheckBehavior := TRUE;
ELSE
	CheckBehavior := FALSE;
END_IF


M_CheckCommand := CheckBehavior;
END_METHOD

METHOD M_CheckUnitsNotBusy : BOOL
VAR_INPUT
END_VAR
M_CheckUnitsNotBusy := true; // need add units check
END_METHOD

METHOD M_CheckUnitsReady : BOOL
VAR_INPUT
END_VAR
M_CheckUnitsReady := NOT (Robot.Error (*OR PullOutConveyor.Error OR FeedInConveyor.bError OR WareHouse.bError*));
END_METHOD

METHOD M_ReloadBox
VAR_INPUT
	Info : ST_FeedInEmptyBox_Info;
END_VAR
IF info.PickUpArea    = E_FeedInEmptyBox_PickUpArea.PullOutConveyorA THEN
    uiExecutingStep   := 1000;
ELSIF info.PickUpArea = E_FeedInEmptyBox_PickUpArea.PullOutConveyorB THEN
    uiExecutingStep   := 2000;
ELSIF info.PickUpArea = E_FeedInEmptyBox_PickUpArea.WareHouseA THEN
    //WareHouse.
ELSIF info.PickUpArea = E_FeedInEmptyBox_PickUpArea.WareHouseB THEN
    uiExecutingStep   := 4000;
ELSE
    _Error := TRUE;
    Status := 'PickUp area value is out of range';
END_IF
END_METHOD

METHOD M_ReloadPulloutConveyorBox : BOOL
VAR_INPUT
	Execute : BOOL;
	SlideSelect : E_PullOutConveyorPosition;
END_VAR
VAR_INST
	uiReloadPulloutConveyorBoxStep : UDINT;
	fbExecute_Rtrig : R_TRIG;
	fbExecute_Ftrig : F_TRIG;
END_VAR
fbExecute_Rtrig(CLK := Execute);
fbExecute_Ftrig(CLK := Execute);
IF fbExecute_Rtrig.Q THEN
	uiReloadPulloutConveyorBoxStep := 100;
ELSIF fbExecute_Ftrig.Q THEN
	uiReloadPulloutConveyorBoxStep := 99000;
END_IF
CASE uiReloadPulloutConveyorBoxStep OF
	0 : 
		// Wait command
	99000:
//		PullOutConveyor.FixCylinderA1.M_MoveBackward('');
//		PullOutConveyor.FixCylinderA2.M_MoveBackward('');
//		PullOutConveyor.FixCylinderB1.M_MoveBackward('');
//		PullOutConveyor.FixCylinderB2.M_MoveBackward('');
END_CASE
END_METHOD

METHOD M_SelectActionMode : E_FeedInAction
VAR_INPUT
END_VAR
IF info.ClampA_Setting.Behavior = E_ClampWork.Work AND info.ClampB_Setting.Behavior <> E_ClampWork.Work THEN
	IF info.ClampA_Setting.PickUpArea = E_FeedInEmptyBox_PickUpArea.WareHouseA THEN
		M_SelectActionMode := E_FeedInAction.ClampA_WareHouseA;
	ELSIF info.ClampA_Setting.PickUpArea = E_FeedInEmptyBox_PickUpArea.WareHouseB THEN
		M_SelectActionMode := E_FeedInAction.ClampA_WareHouseB;
	ELSIF info.ClampA_Setting.PickUpArea = E_FeedInEmptyBox_PickUpArea.PullOutConveyor THEN
		M_SelectActionMode := E_FeedInAction.ClampA_PullOutConveyor;
	END_IF
ELSIF info.ClampA_Setting.Behavior <> E_ClampWork.Work AND info.ClampB_Setting.Behavior = E_ClampWork.Work THEN
	IF info.ClampB_Setting.PickUpArea = E_FeedInEmptyBox_PickUpArea.WareHouseA THEN
		M_SelectActionMode := E_FeedInAction.ClampB_WareHouseA;
	ELSIF info.ClampB_Setting.PickUpArea = E_FeedInEmptyBox_PickUpArea.WareHouseB THEN
		M_SelectActionMode := E_FeedInAction.ClampB_WareHouseB;
	ELSIF info.ClampB_Setting.PickUpArea = E_FeedInEmptyBox_PickUpArea.PullOutConveyor THEN
		M_SelectActionMode := E_FeedInAction.ClampB_PullOutConveyor;
	END_IF
ELSIF info.ClampA_Setting.Behavior = E_ClampWork.Work AND info.ClampB_Setting.Behavior = E_ClampWork.Work THEN
	IF info.ClampA_Setting.PickUpArea = E_FeedInEmptyBox_PickUpArea.PullOutConveyor THEN
		IF  info.ClampB_Setting.PickUpArea = E_FeedInEmptyBox_PickUpArea.WareHouseA THEN
			M_SelectActionMode := E_FeedInAction.A_PullOut_B_WareHouseA;
		ELSIF info.ClampB_Setting.PickUpArea = E_FeedInEmptyBox_PickUpArea.WareHouseB THEN
			M_SelectActionMode := E_FeedInAction.A_PullOut_B_WareHouseB;
		ELSIF info.ClampB_Setting.PickUpArea = E_FeedInEmptyBox_PickUpArea.PullOutConveyor THEN
			M_SelectActionMode := E_FeedInAction.A_PullOut_B_PullOut;
		END_IF
	ELSIF info.ClampA_Setting.PickUpArea = E_FeedInEmptyBox_PickUpArea.WareHouseA THEN
		IF info.ClampB_Setting.PickUpArea = E_FeedInEmptyBox_PickUpArea.WareHouseA THEN
			M_SelectActionMode := E_FeedInAction.A_WareHouseA_B_WareHouseA;
		ELSIF info.ClampB_Setting.PickUpArea = E_FeedInEmptyBox_PickUpArea.WareHouseB THEN
			M_SelectActionMode := E_FeedInAction.A_WareHouseA_B_WareHouseB;
		ELSIF info.ClampB_Setting.PickUpArea = E_FeedInEmptyBox_PickUpArea.PullOutConveyor THEN
			M_SelectActionMode := E_FeedInAction.A_WareHouseA_B_PullOut;
		END_IF
	ELSIF info.ClampA_Setting.PickUpArea = E_FeedInEmptyBox_PickUpArea.WareHouseB THEN
		IF info.ClampB_Setting.PickUpArea = E_FeedInEmptyBox_PickUpArea.WareHouseA THEN
			M_SelectActionMode := E_FeedInAction.A_WareHouseB_B_WareHouseA;
		ELSIF info.ClampB_Setting.PickUpArea = E_FeedInEmptyBox_PickUpArea.WareHouseB THEN
			M_SelectActionMode := E_FeedInAction.A_WareHouseB_B_WareHouseB;
		ELSIF info.ClampB_Setting.PickUpArea = E_FeedInEmptyBox_PickUpArea.PullOutConveyor THEN
			M_SelectActionMode := E_FeedInAction.A_WareHouseB_B_PullOut;
		END_IF
	END_IF
END_IF
END_METHOD

METHOD  M_STATE_ABORTED
VAR_INPUT
END_VAR
Busy    := FALSE;
Aborted := TRUE;
Status := strStatus ;
UniqueErrorCode := _UniqueErrorCode;
IF NOT Execute THEN
    eState := STATE_RESETTING;
END_IF

IF Execute AND Reset THEN
	uiExecutingStep :=uiResumeStep;
	PreviousStrStatus := strStatus;
	PreviousErrorCode := _UniqueErrorCode;
	eState :=STATE_EXECUTING;
END_IF
END_METHOD

METHOD  M_STATE_ABORTING
VAR_INPUT
END_VAR
_AbortCompleted := TRUE;
_Abort :=FALSE;
tonTimeOut.IN:=FALSE;
//DAS.fbStorageArea.M_ResetSlideA_FeedIn();
IF strStatus = PreviousStrStatus THEN
	_UniqueErrorCode :=PreviousErrorCode;
END_IF
IF _AbortCompleted THEN
    eState := STATE_Aborted;
END_IF
END_METHOD

METHOD  M_STATE_DONE
VAR_INPUT
END_VAR
Busy := FALSE;
Done := TRUE;
IF NOT Execute THEN
    eState := STATE_RESETTING;
END_IF
END_METHOD

METHOD  M_STATE_DORMANT
VAR_INPUT
END_VAR
// Clear FB output
Busy            := FALSE;
Done            := FALSE;
Aborted         := FALSE;
Error           :=  FALSE;
ErrorID         := 0;
Status          := '';
_ResetCompleted := FALSE;
_Error          := FALSE;
_Executed       := FALSE;
uiExecutingStep := 0;
uiResettingStep := 0;
uiResumeStep:=0;
tonPlaceSensorDelay.IN :=FALSE;
tonFeedInConveyorDelay.IN :=FALSE;
tonTimeOut.IN :=FALSE;
_UniqueErrorCode :='0';
PreviousStrStatus			 :='';
PreviousErrorCode			 :='';
//DAS.fbStorageArea.M_InactivePulloutConveyorInternCtrl();
// Wait Execute command
IF Execute THEN
    eState := STATE_EXECUTING;
END_IF
END_METHOD

METHOD  M_STATE_ERROR
VAR_INPUT
END_VAR
Robot.Bzone_AllowWork:=FALSE;
IF NOT Execute THEN
    eState := STATE_RESETTING;
END_IF
END_METHOD

METHOD M_STATE_EXECUTING
VAR_INPUT
END_VAR
VAR_INST
    ClampA_WareHouseCoordinates : ST_WareHouseCoordinates;
    ClampB_WareHouseCoordinates : ST_WareHouseCoordinates;
    uiPickUpBothStep            : UINT;
    uiPlaceBothStep             : UINT;
    BoxReady_1st                : BOOL;
    BoxReady_2nd                : BOOL;
    SlideClear_1st              : BOOL;
    SlideClear_2nd              : BOOL;
    TargetWarehouse             : E_WareHouse;
    DiffSizeSlide_Clear         : BOOL;
    SameSizeSlide_clear         : BOOL;
    ActionMode                  : E_FeedInAction;
END_VAR
VAR

END_VAR
// Set status busy
Busy := TRUE;
Robot.Bzone_AllowWork:=Robot._DI12.BzoneInWork;
//Auto mode , just allow robot
IF THIS^.Stop THEN // Pending the timeout when Stop signal occur
	tonTimeout.IN :=FALSE;
END_IF
CASE uiExecutingStep OF
    0:
        // Clear variable
        ActionMode       := E_FeedInAction.Undefined;
        BoxReady_1st     := FALSE;
        BoxReady_2nd     := FALSE;
        uiPickUpBothStep := 0;
        uiPlaceBothStep  := 0;

        // Check command
        IF M_CheckCommand() THEN
            uiExecutingStep := 10;
        END_IF
    10: // Start process, check units first
        IF M_CheckUnitsReady() THEN
            uiExecutingStep := 20;
        END_IF
    20: // Check units not busy state
        IF M_CheckUnitsNotBusy() THEN
            uiExecutingStep := 1000;
        END_IF
    1000:
        // Select action mode
        ActionMode      := M_SelectActionMode();
        uiExecutingStep := 1100;
    1100:
        // according action mode jump step
        CASE ActionMode OF
            E_FeedInAction.ClampA_WareHouseA:
                uiExecutingStep := 10000; // Go to start only ClampA pickup from WareHouseA
            E_FeedInAction.ClampA_WareHouseB:
                uiExecutingStep := 11000; // Go to Start only ClampA pickup from WareHouseB
            E_FeedInAction.ClampA_PullOutConveyor:
                uiExecutingStep := 12000; // Go to Start only ClampA pickup form PulloutConveyor
            E_FeedInAction.ClampB_WareHouseA:
                uiExecutingStep := 20000; // Go to Start only ClampB pickup from WareHouseA
            E_FeedInAction.ClampB_WareHouseB:
                uiExecutingStep := 21000; // Go to Start only ClampB pickup from WareHouseB
            E_FeedInAction.ClampB_PullOutConveyor:
                uiExecutingStep := 22000; // Go to Start only ClampB pickup from PulloutConveyor
            E_FeedInAction.A_WareHouseA_B_WareHouseA:
                uiExecutingStep := 30000; // Go to Start ClampA pickup from WarehouseA, ClampB pickup from WarehouseA
            E_FeedInAction.A_WareHouseA_B_WareHouseB:
                uiExecutingStep := 31000; // Go to Start ClampA pickup from WarehouseA, ClmapB pickup from WarehouseB
            E_FeedInAction.A_WareHouseA_B_PullOut:
                uiExecutingStep := 32000; // Go to Start ClampA pickup from WarehouseA, ClampB pickup from PulloutConveyor
            E_FeedInAction.A_WareHouseB_B_WareHouseA:
                uiExecutingStep := 33000; // Go to Start ClampA pickup from WarehouseB, ClampB pickup from WarehouseA
            E_FeedInAction.A_WareHouseB_B_WareHouseB:
                uiExecutingStep := 34000; // Go to Start ClampA pickup from WarehouseB, CLampB pickup from WarehouseB
            E_FeedInAction.A_WareHouseB_B_PullOut:
                uiExecutingStep := 35000; // Go to Start ClampA pickup from WarehouseB, ClampB pickup from PulloutConveyor
            E_FeedInAction.A_PullOut_B_WareHouseA:
                uiExecutingStep := 36000; // Go to Start ClampA pickup from PulloutConveyor, ClampB pickup from WarehouseA
            E_FeedInAction.A_PullOut_B_WareHouseB:
                uiExecutingStep := 37000; // Go to Start ClampA pickup from PulloutConveyor, ClampB pickup from WarehouseB
            E_FeedInAction.A_PullOut_B_PullOut:
                uiExecutingStep := 38000; // Go to Start ClampBoth pickup from PulloutConveyor
        END_CASE
    10000: // Only clampA pickup box from WareHouseA
        IF NOT Robot._DI1.Done THEN
            ClampA_WareHouseCoordinates := info.ClampA_Setting.WareHouseSetting;
            WareHouse.M_StartReloadBox(WareHouseSelect := E_WareHouse.WareHouseA, WarehouseCoordinates := ClampA_WareHouseCoordinates);

            IF WareHouse.bReloadBox_Completed THEN
                BoxReady_1st := TRUE;
            END_IF

            Robot.M_StartWareHousePickUpBox_ClampA(WareHouseSelect := E_WareHouse.WareHouseA,
                                                   Info            := ClampA_WareHouseCoordinates,
                                                   BoxReady_1st    := BoxReady_1st);
        ELSE
            IF Robot.M_ResetWareHousePickUpBox_ClampA() THEN
                // Clear command and go to place box
				tonTimeOut.IN:=FALSE;
                uiExecutingStep := 60000; // only place clampA
            END_IF
        END_IF
		tonTimeOut.IN :=TRUE;		
		IF tonTimeOut.Q THEN
			tonTimeOut.IN:=FALSE;
			_Error :=TRUE;
			strStatus :='Pick Box timeout';
		END_IF
		
    11000: // Only ClampA pickup box from WareHouseB
        IF NOT Robot._di1.Done THEN
            ClampA_WareHouseCoordinates := info.ClampA_Setting.WareHouseSetting;
            WareHouse.M_StartReloadBox(WareHouseSelect := E_WareHouse.WareHouseB, WarehouseCoordinates := ClampA_WareHouseCoordinates);

            IF WareHouse.bReloadBox_Completed THEN
                BoxReady_1st := TRUE;
            END_IF

            Robot.M_StartWareHousePickUpBox_ClampA(WareHouseSelect := E_WareHouse.WareHouseB,
                                                   Info            := ClampA_WareHouseCoordinates,
                                                   BoxReady_1st    := BoxReady_1st);
        ELSE
            IF Robot.M_ResetWareHousePickUpBox_ClampA() THEN
                // Clear command and go to place box
				tonTimeOut.IN:=FALSE;
                uiExecutingStep := 60000; // only place clampA
            END_IF
        END_IF

		tonTimeOut.IN :=TRUE;		
		IF tonTimeOut.Q THEN
			tonTimeOut.IN:=FALSE;
			_Error :=TRUE;
			strStatus :='Pick Box timeout';
		END_IF
		
    12000: // Only ClampA pickup box from pullout conveyor
        IF NOT Robot._di1.Done THEN
            DAS_CoreSys.MachineControl.fbStorageArea.M_ActivePulloutConveyorInternCtrl();

            IF Info.ClampA_Setting.PullOutConveyorSetting = E_PullOutConveyorAddress.I3_Slide THEN
                DAS_CoreSys.MachineControl.fbStorageArea.M_StartSlideB_FeedIn();
            ELSIF Info.ClampA_Setting.PullOutConveyorSetting = E_PullOutConveyorAddress.I4_Slide THEN
                DAS_CoreSys.MachineControl.fbStorageArea.M_StartSlideA_FeedIn();
            ELSE
                Status := 'Not define PulloutConveyor Slide';
                _Error := TRUE;
            END_IF

            Robot.M_StartPullOutConveyorPickUpBox_ClampA(ClampA_Address := Info.ClampA_Setting.PullOutConveyorSetting,
                                                         BoxReady       := DAS_CoreSys.MachineControl.fballocatearea.fbPulloutCV.Done);
        ELSE
            IF Robot.M_ResetPullOutConveyorPickUpBox_ClampA() THEN
                DAS_CoreSys.MachineControl.fbStorageArea.M_ResetSlideA_FeedIn();
				tonTimeOut.IN:=FALSE;
                uiExecutingStep := 60000; // only place clampA
            END_IF
        END_IF;
			tonTimeOut.IN :=TRUE;		
		IF tonTimeOut.Q THEN
			tonTimeOut.IN:=FALSE;
			_Abort :=TRUE;
			uiResumeStep:=12000;
			strStatus :='Pick Box timeout';
		END_IF
		
    20000: // Only clampB pickup box from WareHouseA
        IF NOT Robot._di1.Done THEN
            ClampB_WareHouseCoordinates := info.ClampB_Setting.WareHouseSetting;
            WareHouse.M_StartReloadBox(WareHouseSelect := E_WareHouse.WareHouseA, WarehouseCoordinates := ClampB_WareHouseCoordinates);

            IF WareHouse.bReloadBox_Completed THEN
                BoxReady_2nd := TRUE;
            END_IF

            Robot.M_StartWareHousePickUpBox_ClampB(WareHouseSelect := E_WareHouse.WareHouseA,
                                                   Info            := ClampB_WareHouseCoordinates,
                                                   BoxReady_2nd    := BoxReady_2nd);
        ELSE
            IF Robot.M_ResetWareHousePickUpBox_ClampB() THEN
                // Clear command and go to place box
				tonTimeOut.IN:=FALSE;
                uiExecutingStep := 70000; // only place clampA
            END_IF
        END_IF
			tonTimeOut.IN :=TRUE;		
		IF tonTimeOut.Q THEN
			tonTimeOut.IN:=FALSE;
			_Error :=TRUE;
			strStatus :='Pick Box timeout';
		END_IF
    21000: // Only ClampB pickup box from WareHouseB
        IF NOT Robot._di1.Done THEN
            ClampB_WareHouseCoordinates := info.ClampB_Setting.WareHouseSetting;
            WareHouse.M_StartReloadBox(WareHouseSelect := E_WareHouse.WareHouseB, WarehouseCoordinates := ClampB_WareHouseCoordinates);

            IF WareHouse.bReloadBox_Completed THEN
                BoxReady_2nd := TRUE;
            END_IF

            Robot.M_StartWareHousePickUpBox_ClampB(WareHouseSelect := E_WareHouse.WareHouseB,
                                                   Info            := ClampB_WareHouseCoordinates,
                                                   BoxReady_2nd    := BoxReady_2nd);
        ELSE
            IF Robot.M_ResetWareHousePickUpBox_ClampB() THEN
                // Clear command and go to place box
				tonTimeOut.IN:=FALSE;
                uiExecutingStep := 70000; // only place clampA
            END_IF
        END_IF
				tonTimeOut.IN :=TRUE;		
		IF tonTimeOut.Q THEN
			tonTimeOut.IN:=FALSE;
			_Error :=TRUE;
			strStatus :='Pick Box timeout';
		END_IF

    22000: // Only ClampB pickup box from PullOut conveyor
        IF NOT Robot._di1.Done THEN
            DAS_CoreSys.MachineControl.fbStorageArea.M_ActivePulloutConveyorInternCtrl();

            IF Info.ClampB_Setting.PullOutConveyorSetting = E_PullOutConveyorAddress.I3_Slide THEN
                DAS_CoreSys.MachineControl.fbStorageArea.M_StartSlideB_FeedIn();
            ELSIF Info.ClampB_Setting.PullOutConveyorSetting = E_PullOutConveyorAddress.I4_Slide THEN
                DAS_CoreSys.MachineControl.fbStorageArea.M_StartSlideA_FeedIn();
            ELSE
                Status := 'Not define PulloutConveyor Slide';
                _Error := TRUE;
            END_IF

            Robot.M_StartPullOutConveyorPickUpBox_ClampB(ClampB_Address := Info.ClampB_Setting.PullOutConveyorSetting,
                                                         BoxReady       := DAS_CoreSys.MachineControl.fballocatearea.fbPulloutCV.Done);
        ELSE
            IF Robot.M_ResetPullOutConveyorPickUpBox_ClampB() THEN
                DAS_CoreSys.MachineControl.fbStorageArea.M_ResetSlideA_FeedIn();
				tonTimeOut.IN:=FALSE;
                uiExecutingStep := 70000; // only place clampA
            END_IF
        END_IF;
			tonTimeOut.IN :=TRUE;		
		IF tonTimeOut.Q THEN
			uiResumeStep:=22000;
			_Abort :=TRUE;
			strStatus :='Pick Box timeout';
		END_IF
		
    30000: // ClampA pickup from WarehouseA, ClampB pickup from WarehouseA
        ClampA_WareHouseCoordinates := info.ClampA_Setting.WareHouseSetting;
        ClampB_WareHouseCoordinates := info.ClampB_Setting.WareHouseSetting;

        CASE uiPickUpBothStep OF
            0: // ClampA target slide move the box to front side
                WareHouse.M_StartReloadBox(WareHouseSelect := E_WareHouse.WareHouseA, WarehouseCoordinates := ClampA_WareHouseCoordinates);

                IF WareHouse.bReloadBox_Completed THEN
                    BoxReady_1st     := TRUE;
                    uiPickUpBothStep := 10;
                END_IF

            10: // wait Robot Allow continue
                IF Robot._DI1.Notification AND
                    NOT
                    WareHouse._stWarehouseList.ASide_Layers[ClampA_WareHouseCoordinates.Layer].stStatus.bSlides[ClampA_WareHouseCoordinates.Slide]
                    THEN
                    WareHouse.M_ResetReloadBox();

                    IF NOT WareHouse.bReloadBox_Completed THEN
                        uiPickUpBothStep := 20;
                    END_IF

                END_IF
            20: // ClampB target slide move the box to front slide
                WareHouse.M_StartReloadBox(WareHouseSelect := E_WareHouse.WareHouseA, WarehouseCoordinates := ClampB_WareHouseCoordinates);

                IF WareHouse.bReloadBox_Completed THEN
                    BoxReady_2nd     := TRUE;
                    uiPickUpBothStep := 99;
                END_IF
            99:
        // wait reset
        END_CASE

        Robot.M_StartWareHousePickUpBox_ClampBoth(WareHouseSelect := E_WareHouse.WareHouseA,
                                                  ClampA_Info     := ClampA_WareHouseCoordinates,
                                                  ClampB_Info     := ClampB_WareHouseCoordinates,
                                                  BoxReady_1st    := BoxReady_1st,
                                                  BoxReady_2nd    := BoxReady_2nd);

        IF Robot._DI1.Done THEN
			tonTimeOut.IN:=FALSE;
            uiExecutingStep := 80000; // go to place step
        END_IF
			tonTimeOut.IN :=TRUE;		
		IF tonTimeOut.Q THEN
			tonTimeOut.IN:=FALSE;
			_Error :=TRUE;
			strStatus :='Pick Box timeout';
		END_IF
		
    31000: // ClampA pickup from WarehouseA, ClampB pickup from WarehouseB
        IF NOT Robot._DI1.Done THEN
            ClampA_WareHouseCoordinates := info.ClampA_Setting.WareHouseSetting;
            WareHouse.M_StartReloadBox(WareHouseSelect := E_WareHouse.WareHouseA, WarehouseCoordinates := ClampA_WareHouseCoordinates);

            IF WareHouse.bReloadBox_Completed THEN
                BoxReady_1st := TRUE;
            END_IF

            Robot.M_StartWareHousePickUpBox_ClampA(WareHouseSelect := E_WareHouse.WareHouseA,
                                                   Info            := ClampA_WareHouseCoordinates,
                                                   BoxReady_1st    := BoxReady_1st);
        ELSE
			tonTimeOut.IN:=FALSE;
			uiExecutingStep := 31080;
		END_IF
			tonTimeOut.IN :=TRUE;		
		IF tonTimeOut.Q THEN
			tonTimeOut.IN:=FALSE;
			_Error :=TRUE;
			strStatus :='Pick Box timeout';
		END_IF
		
	31080:
		Robot.M_ResetAllCommand(); // Clear command and go to place box
		IF NOT Robot._di1.Done THEN
			uiExecutingStep := 31100;// ClampA pickup finished, ClampB pickup start
		END_IF
		
    31100:
        IF NOT Robot._di1.Done THEN
            ClampB_WareHouseCoordinates := info.ClampB_Setting.WareHouseSetting;
            WareHouse.M_StartReloadBox(WareHouseSelect := E_WareHouse.WareHouseB, WarehouseCoordinates := ClampB_WareHouseCoordinates);

            IF WareHouse.bReloadBox_Completed THEN
                BoxReady_2nd := TRUE;
            END_IF

            Robot.M_StartWareHousePickUpBox_ClampB(WareHouseSelect := E_WareHouse.WareHouseB,
                                                   Info            := ClampB_WareHouseCoordinates,
                                                   BoxReady_2nd    := BoxReady_2nd);
        ELSE
			tonTimeOut.IN:=FALSE;
			uiExecutingStep := 31180;
		END_IF
			tonTimeOut.IN :=TRUE;		
		IF tonTimeOut.Q THEN
			tonTimeOut.IN:=FALSE;
			_Error :=TRUE;
			strStatus :='Pick Box timeout';
		END_IF
		
	31180:
		Robot.M_ResetAllCommand(); // Clear command and go to place box
		IF NOT Robot._di1.Done THEN
			uiExecutingStep := 80000;// ClampA pickup finished, ClampB pickup start
		END_IF
    32000: // ClampA pickup from WarehouseA, ClampB pickup from PulloutConveyor
        IF NOT Robot._DI1.Done THEN
            ClampA_WareHouseCoordinates := info.ClampA_Setting.WareHouseSetting;
            WareHouse.M_StartReloadBox(WareHouseSelect := E_WareHouse.WareHouseA, WarehouseCoordinates := ClampA_WareHouseCoordinates);

            IF WareHouse.bReloadBox_Completed THEN
                BoxReady_1st := TRUE;
            END_IF

            Robot.M_StartWareHousePickUpBox_ClampA(WareHouseSelect := E_WareHouse.WareHouseA,
                                                   Info            := ClampA_WareHouseCoordinates,
                                                   BoxReady_1st    := BoxReady_1st);
        ELSE
			tonTimeOut.IN:=FALSE;
			uiExecutingStep := 32080; // ClampA pickup finished, ClampB start	
        END_IF
			tonTimeOut.IN :=TRUE;		
		IF tonTimeOut.Q THEN
			tonTimeOut.IN:=FALSE;
			_Error :=TRUE;
			strStatus :='Pick Box timeout';
		END_IF
	32080:
		Robot.M_ResetAllCommand();
		// Clear command and go to place box
		IF NOT Robot._di1.Done THEN
			uiExecutingStep := 32100;// ClampA pickup finished, ClampB start
		END_IF
    32100:
        IF NOT Robot._di1.Done THEN
        DAS_CoreSys.MachineControl.fballocatearea.M_GetPulloutAccess(ControlAccess := E_RoundBeltControlAccess.FanucRobot);

            IF Info.ClampB_Setting.PullOutConveyorSetting = E_PullOutConveyorAddress.I3_Slide THEN
                        DAS_CoreSys.MachineControl.fballocatearea
                            .M_StartStoragePulloutAction(CommandType := E_PullOutConveyorCommandType.SlideB_FeedIn_Ext,
                                                         CV_BackwardTIme := T#0S,
                                                         CV_ForwardTime := T#0S);
            ELSIF Info.ClampB_Setting.PullOutConveyorSetting = E_PullOutConveyorAddress.I4_Slide THEN
                        DAS_CoreSys.MachineControl.fballocatearea
                            .M_StartStoragePulloutAction(CommandType := E_PullOutConveyorCommandType.SlideA_FeedIn_Ext,
                                                         CV_BackwardTIme := T#0S,
                                                         CV_ForwardTime := T#0S);
            ELSE
                Status := 'Not define PulloutConveyor Slide';
                _Error := TRUE;
            END_IF

            Robot.M_StartPullOutConveyorPickUpBox_ClampB(ClampB_Address := Info.ClampB_Setting.PullOutConveyorSetting,
                                                         BoxReady       := DAS_CoreSys.MachineControl.fballocatearea.fbPulloutCV.Done);
        ELSE
			tonTimeOut.IN:=FALSE;
			uiExecutingStep := 32180;
		END_IF
			tonTimeOut.IN :=TRUE;		
		IF tonTimeOut.Q THEN
			tonTimeOut.IN:=FALSE;
			_Error :=TRUE;
			strStatus :='Pick Box timeout';
		END_IF
	32180:
		robot.M_ResetAllCommand();
		IF NOT Robot._DI1.Done THEN
			uiExecutingStep := 80000;
		END_IF
    33000: // ClampA Pickup from WarehouseB, ClampB pickup from WarehouseA
        IF NOT Robot._di1.Done THEN
            ClampA_WareHouseCoordinates := info.ClampA_Setting.WareHouseSetting;
            WareHouse.M_StartReloadBox(WareHouseSelect := E_WareHouse.WareHouseB, WarehouseCoordinates := ClampA_WareHouseCoordinates);

            IF WareHouse.bReloadBox_Completed THEN
                BoxReady_1st := TRUE;
            END_IF

            Robot.M_StartWareHousePickUpBox_ClampA(WareHouseSelect := E_WareHouse.WareHouseB,
                                                   Info            := ClampA_WareHouseCoordinates,
                                                   BoxReady_1st    := BoxReady_1st);
        ELSE
			tonTimeOut.IN:=FALSE;
			uiExecutingStep := 33080;
		END_IF
				tonTimeOut.IN :=TRUE;		
		IF tonTimeOut.Q THEN
			tonTimeOut.IN:=FALSE;
			_Error :=TRUE;
			strStatus :='Pick Box timeout';
		END_IF
	33080:
		Robot.M_ResetAllCommand(); // Clear command and go to place box
		IF NOT Robot._DI1.Done THEN
                uiExecutingStep := 33100; // only place clampA
        END_IF
    33100:
        IF NOT Robot._di1.Done THEN
            ClampB_WareHouseCoordinates := info.ClampB_Setting.WareHouseSetting;
            WareHouse.M_StartReloadBox(WareHouseSelect := E_WareHouse.WareHouseA, WarehouseCoordinates := ClampB_WareHouseCoordinates);

            IF WareHouse.bReloadBox_Completed THEN
                BoxReady_2nd := TRUE;
            END_IF

            Robot.M_StartWareHousePickUpBox_ClampB(WareHouseSelect := E_WareHouse.WareHouseA,
                                                   Info            := ClampB_WareHouseCoordinates,
                                                   BoxReady_2nd    := BoxReady_2nd);
        ELSE
			Robot.M_ResetAllCommand(); // Clear command and go to place box
			IF NOT Robot._DI1.Done THEN
				tonTimeOut.IN:=FALSE;
				uiExecutingStep := 80000; // only place clampA
			END_IF
        END_IF
		tonTimeOut.IN :=TRUE;		
		IF tonTimeOut.Q THEN
			tonTimeOut.IN:=FALSE;
			_Error :=TRUE;
			strStatus :='Place Box timeout';
		END_IF
		
    34000: // ClampA pickup from WarehouseB, ClampB pickup from WarehouseB
        ClampA_WareHouseCoordinates := info.ClampA_Setting.WareHouseSetting;
        ClampB_WareHouseCoordinates := info.ClampB_Setting.WareHouseSetting;

        CASE uiPickUpBothStep OF
            0: // ClampA target slide move the box to front side
                WareHouse.M_StartReloadBox(WareHouseSelect := E_WareHouse.WareHouseB, WarehouseCoordinates := ClampA_WareHouseCoordinates);

                IF WareHouse.bReloadBox_Completed THEN
                    BoxReady_1st     := TRUE;
                    uiPickUpBothStep := 10;
                END_IF

            10: // wait Robot Allow continue
                IF Robot._DI1.Notification AND
                    NOT
                    WareHouse._stWarehouseList.BSide_Layers[ClampA_WareHouseCoordinates.Layer].stStatus.bSlides[ClampA_WareHouseCoordinates.Slide]
                    THEN
                    WareHouse.M_ResetReloadBox();

                    IF NOT WareHouse.bReloadBox_Completed THEN
                        uiPickUpBothStep := 20;
                    END_IF

                END_IF
            20: // ClampB target slide move the box to front slide
                WareHouse.M_StartReloadBox(WareHouseSelect := E_WareHouse.WareHouseB, WarehouseCoordinates := ClampB_WareHouseCoordinates);

                IF WareHouse.bReloadBox_Completed THEN
                    BoxReady_2nd     := TRUE;
                    uiPickUpBothStep := 99;
                END_IF
            99:
        // wait reset
        END_CASE

        Robot.M_StartWareHousePickUpBox_ClampBoth(WareHouseSelect := E_WareHouse.WareHouseB,
                                                  ClampA_Info     := ClampA_WareHouseCoordinates,
                                                  ClampB_Info     := ClampB_WareHouseCoordinates,
                                                  BoxReady_1st    := BoxReady_1st,
                                                  BoxReady_2nd    := BoxReady_2nd);

        IF Robot._DI1.Done THEN
			tonTimeOut.IN:=FALSE;
            uiExecutingStep := 80000; // go to place step
        END_IF
		
			tonTimeOut.IN :=TRUE;		
		IF tonTimeOut.Q THEN
			tonTimeOut.IN:=FALSE;
			_Error :=TRUE;
			strStatus :='Pick Box timeout';
		END_IF
		
    35000: // ClampA pickup from WarehouseB, ClampB pickup from PulloutConveyor
        IF NOT Robot._di1.Done THEN
        DAS_CoreSys.MachineControl.fballocatearea.M_GetPulloutAccess(ControlAccess := E_RoundBeltControlAccess.FanucRobot);

            IF Info.ClampA_Setting.PullOutConveyorSetting = E_PullOutConveyorAddress.I3_Slide THEN
                        DAS_CoreSys.MachineControl.fballocatearea
                            .M_StartStoragePulloutAction(CommandType := E_PullOutConveyorCommandType.SlideB_FeedIn_Ext,
                                                         CV_BackwardTIme := T#0S,
                                                         CV_ForwardTime := T#0S);
            ELSIF Info.ClampA_Setting.PullOutConveyorSetting = E_PullOutConveyorAddress.I4_Slide THEN
                        DAS_CoreSys.MachineControl.fballocatearea
                            .M_StartStoragePulloutAction(CommandType := E_PullOutConveyorCommandType.SlideA_FeedIn_Ext,
                                                         CV_BackwardTIme := T#0S,
                                                         CV_ForwardTime := T#0S);
            ELSE
                Status := 'Not define PulloutConveyor Slide';
                _Error := TRUE;
            END_IF

            Robot.M_StartPullOutConveyorPickUpBox_ClampA(ClampA_Address := Info.ClampA_Setting.PullOutConveyorSetting,
                                                         BoxReady       := DAS_CoreSys.MachineControl.fballocatearea.fbPulloutCV.Done);
        ELSE
            IF Robot.M_ResetPullOutConveyorPickUpBox_ClampA() THEN
            DAS_CoreSys.MachineControl.fballocatearea.M_StopStoragePulloutAction();
				tonTimeOut.IN:=FALSE;
                uiExecutingStep := 35100; // only place clampA
            END_IF
        END_IF;
			tonTimeOut.IN :=TRUE;		
		IF tonTimeOut.Q THEN
			tonTimeOut.IN:=FALSE;
			_Error :=TRUE;
			strStatus :='Pick Box timeout';
		END_IF
		
    35100:
        IF NOT Robot._di1.Done THEN
        DAS_CoreSys.MachineControl.fballocatearea.M_GetPulloutAccess(ControlAccess := E_RoundBeltControlAccess.FanucRobot);

            IF Info.ClampB_Setting.PullOutConveyorSetting = E_PullOutConveyorAddress.I3_Slide THEN
                        DAS_CoreSys.MachineControl.fballocatearea
                            .M_StartStoragePulloutAction(CommandType := E_PullOutConveyorCommandType.SlideB_FeedIn_Ext,
                                                         CV_BackwardTIme := T#0S,
                                                         CV_ForwardTime := T#0S);
            ELSIF Info.ClampB_Setting.PullOutConveyorSetting = E_PullOutConveyorAddress.I4_Slide THEN
                        DAS_CoreSys.MachineControl.fballocatearea
                            .M_StartStoragePulloutAction(CommandType := E_PullOutConveyorCommandType.SlideA_FeedIn_Ext,
                                                         CV_BackwardTIme := T#0S,
                                                         CV_ForwardTime := T#0S);
            ELSE
                Status := 'Not define PulloutConveyor Slide';
                _Error := TRUE;
            END_IF

            Robot.M_StartPullOutConveyorPickUpBox_ClampB(ClampB_Address := Info.ClampB_Setting.PullOutConveyorSetting,
                                                         BoxReady       := DAS_CoreSys.MachineControl.fballocatearea.fbPulloutCV.Done);
        ELSE
            IF Robot.M_ResetPullOutConveyorPickUpBox_ClampB() THEN
            DAS_CoreSys.MachineControl.fballocatearea.M_StopStoragePulloutAction();
				tonTimeOut.IN:=FALSE;
                uiExecutingStep := 80000; // only place clampA
            END_IF
        END_IF;
				tonTimeOut.IN :=TRUE;		
		IF tonTimeOut.Q THEN
			tonTimeOut.IN:=FALSE;
			_Error :=TRUE;
			strStatus :='Pick Box timeout';
		END_IF
		
    36000: // ClampA pickup from PulloutConveyor, ClampB pickup from WarehouseA
        IF NOT Robot._di1.Done THEN
        DAS_CoreSys.MachineControl.fballocatearea.M_GetPulloutAccess(ControlAccess := E_RoundBeltControlAccess.FanucRobot);

            IF Info.ClampA_Setting.PullOutConveyorSetting = E_PullOutConveyorAddress.I3_Slide THEN
                        DAS_CoreSys.MachineControl.fballocatearea
                            .M_StartStoragePulloutAction(CommandType := E_PullOutConveyorCommandType.SlideB_FeedIn_Ext,
                                                         CV_BackwardTIme := T#0S,
                                                         CV_ForwardTime := T#0S);
            ELSIF Info.ClampA_Setting.PullOutConveyorSetting = E_PullOutConveyorAddress.I4_Slide THEN
                        DAS_CoreSys.MachineControl.fballocatearea
                            .M_StartStoragePulloutAction(CommandType := E_PullOutConveyorCommandType.SlideA_FeedIn_Ext,
                                                         CV_BackwardTIme := T#0S,
                                                         CV_ForwardTime := T#0S);
            ELSE
                Status := 'Not define PulloutConveyor Slide';
                _Error := TRUE;
            END_IF

            Robot.M_StartPullOutConveyorPickUpBox_ClampA(ClampA_Address := Info.ClampA_Setting.PullOutConveyorSetting,
                                                         BoxReady       := DAS_CoreSys.MachineControl.fballocatearea.fbPulloutCV.Done);
        ELSE
			tonTimeOut.IN:=FALSE;
			uiExecutingStep := 36080;
		END_IF
				tonTimeOut.IN :=TRUE;		
		IF tonTimeOut.Q THEN
			tonTimeOut.IN:=FALSE;
			_Error :=TRUE;
			strStatus :='Pick Box timeout';
		END_IF
		
	36080:
		Robot.M_ResetAllCommand();
        DAS_CoreSys.MachineControl.fballocatearea.M_StopStoragePulloutAction();
		IF NOT Robot._di1.Done THEN
			uiExecutingStep := 36100; // only place clampA
		END_IF
    36100:
        IF NOT Robot._di1.Done THEN
            ClampB_WareHouseCoordinates := info.ClampB_Setting.WareHouseSetting;
            WareHouse.M_StartReloadBox(WareHouseSelect := E_WareHouse.WareHouseA, WarehouseCoordinates := ClampB_WareHouseCoordinates);

            IF WareHouse.bReloadBox_Completed THEN
                BoxReady_2nd := TRUE;
            END_IF

            Robot.M_StartWareHousePickUpBox_ClampB(WareHouseSelect := E_WareHouse.WareHouseA,
                                                   Info            := ClampB_WareHouseCoordinates,
                                                   BoxReady_2nd    := BoxReady_2nd);
        ELSE
			tonTimeOut.IN:=FALSE;
			uiExecutingStep := 36200;
		END_IF
				tonTimeOut.IN :=TRUE;		
		IF tonTimeOut.Q THEN
			tonTimeOut.IN:=FALSE;
			_Error :=TRUE;
			strStatus :='Pick Box timeout';
		END_IF
		
	36200:
		Robot.M_ResetAllCommand(); // Clear command and go to place box
		IF NOT Robot._DI1.Done THEN
			uiExecutingStep := 80000; //  place clampA and clampB
		END_IF 
    37000: // ClampA pickup from PulloutConveyor, ClampB pickup from WarehouseB
        IF NOT Robot._di1.Done THEN
        DAS_CoreSys.MachineControl.fballocatearea.M_GetPulloutAccess(ControlAccess := E_RoundBeltControlAccess.FanucRobot);

            IF Info.ClampA_Setting.PullOutConveyorSetting = E_PullOutConveyorAddress.I3_Slide THEN
                        DAS_CoreSys.MachineControl.fballocatearea
                            .M_StartStoragePulloutAction(CommandType := E_PullOutConveyorCommandType.SlideB_FeedIn_Ext,
                                                         CV_BackwardTIme := T#0S,
                                                         CV_ForwardTime := T#0S);
            ELSIF Info.ClampA_Setting.PullOutConveyorSetting = E_PullOutConveyorAddress.I4_Slide THEN
                        DAS_CoreSys.MachineControl.fballocatearea
                            .M_StartStoragePulloutAction(CommandType := E_PullOutConveyorCommandType.SlideA_FeedIn_Ext,
                                                         CV_BackwardTIme := T#0S,
                                                         CV_ForwardTime := T#0S);
            ELSE
                Status := 'Not define PulloutConveyor Slide';
                _Error := TRUE;
            END_IF

            Robot.M_StartPullOutConveyorPickUpBox_ClampA(ClampA_Address := Info.ClampA_Setting.PullOutConveyorSetting,
                                                         BoxReady       := DAS_CoreSys.MachineControl.fballocatearea.fbPulloutCV.Done);
        ELSE
			tonTimeOut.IN:=FALSE;
			uiExecutingStep := 37080;
		END_IF
					tonTimeOut.IN :=TRUE;		
		IF tonTimeOut.Q THEN
			tonTimeOut.IN:=FALSE;
			_Error :=TRUE;
			strStatus :='Pick Box timeout';
		END_IF
		
		
	37080:
		Robot.M_ResetAllCommand();
		IF NOT Robot._di1.Done THEN
			// Clear Pullout conveyor reload command
            DAS_CoreSys.MachineControl.fballocatearea.M_StopStoragePulloutAction();
			uiExecutingStep := 37100;
		END_IF
    37100:
        IF NOT Robot._di1.Done THEN
            ClampB_WareHouseCoordinates := info.ClampB_Setting.WareHouseSetting;
            WareHouse.M_StartReloadBox(WareHouseSelect := E_WareHouse.WareHouseB, WarehouseCoordinates := ClampB_WareHouseCoordinates);

            IF WareHouse.bReloadBox_Completed THEN
                BoxReady_2nd := TRUE;
            END_IF

            Robot.M_StartWareHousePickUpBox_ClampB(WareHouseSelect := E_WareHouse.WareHouseB,
                                                   Info            := ClampB_WareHouseCoordinates,
                                                   BoxReady_2nd    := BoxReady_2nd);
        ELSE
			tonTimeOut.IN:=FALSE;
			uiExecutingStep := 37180;
		END_IF
		tonTimeOut.IN :=TRUE;		
		IF tonTimeOut.Q THEN
			tonTimeOut.IN:=FALSE;
			_Error :=TRUE;
			strStatus :='Pick Box timeout';
		END_IF
	37180:
		Robot.M_ResetAllCommand(); // Clear command and go to place box
		IF NOT Robot._di1.Done THEN
			uiExecutingStep := 80000; // only place clampA
		END_IF
    38000: // ClampBoth pickup from PulloutConveyor
        DAS_CoreSys.MachineControl.fballocatearea.M_GetPulloutAccess(ControlAccess := E_RoundBeltControlAccess.FanucRobot);

        CASE uiPickUpBothStep OF
            0: // ClampA target slide move the box to front side
                IF Info.ClampA_Setting.PullOutConveyorSetting = E_PullOutConveyorAddress.I3_Slide THEN
                        DAS_CoreSys.MachineControl.fballocatearea
                            .M_StartStoragePulloutAction(CommandType := E_PullOutConveyorCommandType.SlideB_FeedIn_Ext,
                                                         CV_BackwardTIme := T#0S,
                                                         CV_ForwardTime := T#0S);
                ELSIF Info.ClampA_Setting.PullOutConveyorSetting = E_PullOutConveyorAddress.I4_Slide THEN
                        DAS_CoreSys.MachineControl.fballocatearea
                            .M_StartStoragePulloutAction(CommandType := E_PullOutConveyorCommandType.SlideA_FeedIn_Ext,
                                                         CV_BackwardTIme := T#0S,
                                                         CV_ForwardTime := T#0S);
                ELSE
                    Status := 'Not define PulloutConveyor Slide';
                    _Error := TRUE;
                END_IF

                IF DAS_CoreSys.MachineControl.fballocatearea.fbpulloutcv.Done THEN
                    BoxReady_1st     := TRUE;
                    uiPickUpBothStep := 10;
                END_IF

            10: // wait Robot Allow continue
                IF Robot._DI1.Notification THEN
            		DAS_CoreSys.MachineControl.fballocatearea.M_StopStoragePulloutAction();

                    IF NOT DAS_CoreSys.MachineControl.fballocatearea.fbpulloutcv.Done THEN
                        uiPickUpBothStep := 20;
                    END_IF

                END_IF
            20: // ClampB target slide move the box to front slide
                IF Info.ClampB_Setting.PullOutConveyorSetting = E_PullOutConveyorAddress.I3_Slide THEN
                        DAS_CoreSys.MachineControl.fballocatearea
                            .M_StartStoragePulloutAction(CommandType := E_PullOutConveyorCommandType.SlideB_FeedIn_Ext,
                                                         CV_BackwardTIme := T#0S,
                                                         CV_ForwardTime := T#0S);
                ELSIF Info.ClampB_Setting.PullOutConveyorSetting = E_PullOutConveyorAddress.I4_Slide THEN
                        DAS_CoreSys.MachineControl.fballocatearea
                            .M_StartStoragePulloutAction(CommandType := E_PullOutConveyorCommandType.SlideA_FeedIn_Ext,
                                                         CV_BackwardTIme := T#0S,
                                                         CV_ForwardTime := T#0S);
                ELSE
                    Status := 'Not define PulloutConveyor Slide';
                    _Error := TRUE;
                END_IF

                IF DAS_CoreSys.MachineControl.fballocatearea.fbpulloutcv.Done THEN
                    BoxReady_2nd     := TRUE;
                    uiPickUpBothStep := 99;
                END_IF
            99:
        // wait reset
        END_CASE

        Robot.M_StartPullOutConveyorPickUpBox_ClampBoth(ClampA_Address := Info.ClampA_Setting.PullOutConveyorSetting,
                                                        ClampB_Address := Info.ClampB_Setting.PullOutConveyorSetting,
                                                        BoxReady_1     := BoxReady_1st,
                                                        BoxReady_2     := BoxReady_2nd);

        IF Robot._DI1.Done THEN
			tonTimeOut.IN:=FALSE;
            uiExecutingStep := 80000; // go to place step
        END_IF
		
		tonTimeOut.IN :=TRUE;		
		IF tonTimeOut.Q THEN
			tonTimeOut.IN:=FALSE;
			_Abort :=TRUE;	
			uiResumeStep:=38000;		
			strStatus :='Pick Box timeout';
		END_IF
    60000: // Only ClampA place box
        // Clear command
        WareHouse.M_ResetReloadBox();
        Robot.M_ResetAllCommand();

        // Check robot RSR1 not working
        IF NOT Robot._DI1.Done AND NOT (Robot._DI1.AbsMoveA OR Robot._DI1.AbsMoveB OR Robot._DI1.WarehouseA OR Robot._DI1.WarehouseB) THEN
            uiExecutingStep := 61000;
        END_IF
    61000: // Only ClampA place box Start
        IF NOT Robot._DI1.Done THEN
			IF NOT DiffSizeCV.InBackWard AND SameSizeCV.InBackWard THEN
				CASE Info.ClampA_Setting.PlaceArea OF
					E_FeedInEmptyBox_PlaceArea.DiffSizeConveyor:
					
            			DiffSizeCV.M_MoveForward();
					E_FeedInEmptyBox_PlaceArea.SameSizeConveyor:
						SameSizeCV.M_MoveForward();
				END_CASE

            	IF Input.bDifferentSizeCV_BoxDetect7_Sensor THEN
                	DiffSizeSlide_Clear := FALSE;
            	ELSE
                	DiffSizeSlide_Clear := TRUE;
            	END_IF

            	IF Input.bSameSizeCV_BoxNearStorageSensor THEN
                	SameSizeSlide_clear := FALSE;
            	ELSE
                	SameSizeSlide_clear := TRUE;
            	END_IF
			ELSE
					DiffSizeSlide_Clear := FALSE;
					SameSizeSlide_clear := FALSE;	
			END_IF
			
            Robot.M_StartMoveBoxToFeedInConveyor_ClampA(ConveyorSlideSelect := Info.ClampA_Setting.PlaceArea,
                                                        DiffSizeSlideClear  := DiffSizeSlide_Clear,
                                                        SameSizeSlideClear  := SameSizeSlide_clear);
        ELSE
			tonTimeOut.IN:=FALSE;
            uiExecutingStep := 99000; // Go to process end
        END_IF
		tonTimeOut.IN :=TRUE;		
		IF tonTimeOut.Q THEN
			tonTimeOut.IN:=FALSE;
			_Abort :=TRUE;		
			uiResumeStep:=61000;	
			strStatus :='Place Box timeout';
		END_IF
    70000: // Only ClampB place box
        // Clear command
        WareHouse.M_ResetReloadBox();
        Robot.M_ResetAllCommand();

        // Check robot RSR1 not working
        IF NOT Robot._DI1.Done AND NOT (Robot._DI1.AbsMoveA OR Robot._DI1.AbsMoveB OR Robot._DI1.WarehouseA OR Robot._DI1.WarehouseB) THEN
            uiExecutingStep := 71000;
        END_IF
    71000:
        IF NOT Robot._DI1.Done THEN
			IF NOT DiffSizeCV.InBackWard AND SameSizeCV.InBackWard THEN
				CASE Info.ClampA_Setting.PlaceArea OF
					E_FeedInEmptyBox_PlaceArea.DiffSizeConveyor:
					
            			DiffSizeCV.M_MoveForward();
					E_FeedInEmptyBox_PlaceArea.SameSizeConveyor:
						SameSizeCV.M_MoveForward();
				END_CASE

    	        IF input.bDifferentSizeCV_BoxDetect7_Sensor THEN
        	        DiffSizeSlide_Clear := FALSE;
            	ELSE
                	DiffSizeSlide_Clear := TRUE;
            	END_IF

            	IF Input.bSameSizeCV_BoxNearStorageSensor THEN
                	SameSizeSlide_clear := FALSE;
            	ELSE
            	    SameSizeSlide_clear := TRUE;
          	  END_IF
			ELSE
					DiffSizeSlide_Clear := FALSE;
					SameSizeSlide_clear := FALSE;	
			END_IF
            Robot.M_StartMoveBoxToFeedInConveyor_ClampB(ConveyorSlideSelect := Info.ClampB_Setting.PlaceArea,
                                                        DiffSizeSlideClear  := DiffSizeSlide_Clear,
                                                        SameSizeSlideClear  := SameSizeSlide_clear);
        ELSE
			tonTimeOut.IN:=FALSE;
            uiExecutingStep := 99000; // Go to process end
        END_IF
		tonTimeOut.IN :=TRUE;		
		IF tonTimeOut.Q THEN
			tonTimeOut.IN:=FALSE;
			_Abort :=TRUE;		
			uiResumeStep:=71000;	
			strStatus :='Place Box timeout';
		END_IF
    80000: // Both Clamp place box
        WareHouse.M_ResetReloadBox(); // Clear Warehouse reload command
        Robot.M_ResetAllCommand(); // Clear Fanuc Robot command
        IF NOT Robot._DI1.Done THEN
            uiExecutingStep := 81000;
        END_IF;
    81000:
			
        CASE uiPlaceBothStep OF
			
            0:                
                SlideClear_1st  := FALSE;
                SlideClear_2nd  := FALSE;
			IF NOT DiffSizeCV.InBackWard AND NOT SameSizeCV.InBackWard THEN
				CASE Info.ClampA_Setting.PlaceArea OF
					E_FeedInEmptyBox_PlaceArea.DiffSizeConveyor:
            			DiffSizeCV.M_MoveForward();
						uiPlaceBothStep := 10;
					E_FeedInEmptyBox_PlaceArea.SameSizeConveyor:
						SameSizeCV.M_MoveForward();
						uiPlaceBothStep := 10;
				END_CASE
			END_IF
            10:
                // ClampA place box
				
				CASE Info.ClampA_Setting.PlaceArea OF
					E_FeedInEmptyBox_PlaceArea.DiffSizeConveyor:
						IF NOT DiffSizeCV.InStopped  THEN
							DiffSizeCV.M_MoveForward();
						END_IF
						//uiPlaceBothStep := 10;
					E_FeedInEmptyBox_PlaceArea.SameSizeConveyor:
						IF  NOT SameSizeCV.InStopped  THEN
							SameSizeCV.M_MoveForward();
						END_IF
						//uiPlaceBothStep := 10;
				END_CASE

				
				IF	NOT DiffSizeCV.InStopped OR  NOT SameSizeCV.InStopped THEN
                	IF info.ClampA_Setting.PlaceArea = E_FeedInEmptyBox_PlaceArea.DiffSizeConveyor THEN
                    	IF Input.bDifferentSizeCV_BoxDetect7_Sensor THEN
                        	SlideClear_1st := FALSE;
                    	ELSE
                        	SlideClear_1st := TRUE;
                    	END_IF

                	ELSIF info.ClampA_Setting.PlaceArea = E_FeedInEmptyBox_PlaceArea.SameSizeConveyor THEN
                    	IF Input.bSameSizeCV_BoxNearStorageSensor THEN
                        	SlideClear_1st := FALSE;
                    	ELSE
                        	SlideClear_1st := TRUE;
                    	END_IF
                	END_IF
					IF SlideClear_1st AND NOT Robot._di1.ClampA_Sensor THEN
                		uiPlaceBothStep := 20;
					END_IF
				ELSE
					SlideClear_1st := FALSE;
				END_IF
            20:
				SlideClear_2nd := FALSE;
				tonPlaceSensorDelay.IN :=FALSE;
				IF NOT DiffSizeCV.InStopped THEN
					DiffSizeCV.M_MoveForward();
				END_IF
				IF NOT SameSizeCV.InStopped THEN
					SameSizeCV.M_MoveForward();
				END_IF
                IF ((info.ClampA_Setting.PlaceArea = E_FeedInEmptyBox_PlaceArea.DiffSizeConveyor) AND NOT Input.bDifferentSizeCV_BoxDetect7_Sensor) THEN
					 uiPlaceBothStep := 30;
                ELSIF ((info.ClampA_Setting.PlaceArea = E_FeedInEmptyBox_PlaceArea.SameSizeConveyor) AND NOT Input.bSameSizeCV_BoxDetect6_Sensor) THEN
                     uiPlaceBothStep := 30;
                END_IF
            30:
                // ClampB place box
				CASE Info.ClampB_Setting.PlaceArea OF
					E_FeedInEmptyBox_PlaceArea.DiffSizeConveyor:
						IF   DiffSizeCV.InStopped  THEN
							DiffSizeCV.M_MoveForward();
						END_IF
						//uiPlaceBothStep := 10;
					E_FeedInEmptyBox_PlaceArea.SameSizeConveyor:
						IF   SameSizeCV.InStopped  THEN
							SameSizeCV.M_MoveForward();
						END_IF
						//uiPlaceBothStep := 10;
				END_CASE
				IF	 NOT DiffSizeCV.InStopped OR NOT SameSizeCV.InStopped THEN
               		 IF info.ClampB_Setting.PlaceArea = E_FeedInEmptyBox_PlaceArea.DiffSizeConveyor THEN
                 	   IF Input.bDifferentSizeCV_BoxDetect7_Sensor THEN
						
                    	    SlideClear_2nd := FALSE;
                   		 ELSE                        
							tonPlaceSensorDelay.IN :=TRUE	;
								IF tonPlaceSensorDelay.Q THEN
									SlideClear_2nd := TRUE;
								END_IF
                   		 END_IF
					
               		 ELSIF info.ClampB_Setting.PlaceArea = E_FeedInEmptyBox_PlaceArea.SameSizeConveyor THEN
                 	   IF Input.bSameSizeCV_BoxNearStorageSensor THEN
                 	       SlideClear_2nd := FALSE;
                 	   ELSE
                        
							tonPlaceSensorDelay.IN :=TRUE	;
								IF tonPlaceSensorDelay.Q THEN
							SlideClear_2nd := TRUE;
								END_IF
                  		 END_IF
               			 END_IF
				END_IF
				
				IF SlideClear_2nd THEN
                	uiPlaceBothStep := 99;
					tonPlaceSensorDelay.IN :=FALSE;
				END_IF
			
            99:
        // wait reset
        END_CASE

        IF NOT Robot._DI1.Done THEN
            Robot.M_StartMoveBoxToFeedInConveyor_ClampBoth(ClampA_Address := info.ClampA_Setting.PlaceArea,
                                                           ClampB_Address := info.ClampB_Setting.PlaceArea,
                                                           SlideClear_1st := SlideClear_1st,
                                                           SlideClear_2nd := SlideClear_2nd);
        ELSE
			tonTimeOut.IN:=FALSE;
            uiExecutingStep := 99000;
        END_IF
		tonTimeOut.IN :=TRUE;		
		IF tonTimeOut.Q THEN
			tonTimeOut.IN:=FALSE;
			_Abort :=TRUE;	
			uiResumeStep:=81000;		
			strStatus :='Place Box timeout';
		END_IF
    99000: // process done
        // Stop FeedIn conveyor
		tonFeedInConveyorDelay.IN :=TRUE;		//Delay FeedInConveyor stop 500MS Edit by Min
		IF tonFeedInConveyorDelay.Q THEN
			DAS_CoreSys.MachineControl.fballocatearea.M_ReleasePulloutAccess(ControlAccess := E_RoundBeltControlAccess.FanucRobot);
			DiffSizeCV.M_MotorStop();
			SameSizeCV.M_MotorStop();
			tonFeedInConveyorDelay.IN :=FALSE;
			Status    := 'Process completed';
				IF DiffSizeCV.InStopped AND SameSizeCV.InStopped THEN
				 _Executed := TRUE;
				END_IF
		END_IF
END_CASE

IF _Executed THEN
    eState := STATE_DONE;
ELSIF NOT Execute THEN
    eState := STATE_RESETTING;
ELSIF Abort OR _Abort THEN
	//FUN_UniqueErrorCodeGenerator(iErrorID := ErrorID,UinqueErrorCode=>_UniqueErrorCode);
	eState := STATE_ABORTING;
ELSIF _Error THEN
	//FUN_UniqueErrorCodeGenerator(iErrorID := ErrorID,UinqueErrorCode=>_UniqueErrorCode);
	eState := STATE_ERROR;
	
END_IF
END_METHOD

METHOD  M_STATE_RESETTING
VAR_INPUT
END_VAR
IF _Executed THEN Done :=TRUE ; END_IF
CASE uiResettingStep OF
	0:
		//DAS.fbStorageArea.M_InactivePulloutConveyorInternCtrl();
		Robot.M_ResetAllCommand();
		Robot.Bzone_AllowWork:=FALSE;
		DiffSizeCV.M_MotorStop();
		SameSizeCV.M_MotorStop();
		 DAS_CoreSys.MachineControl.fballocatearea.M_ReleasePulloutAccess(ControlAccess := E_RoundBeltControlAccess.FanucRobot);
		 DAS_CoreSys.MachineControl.fballocatearea.M_StopStoragePulloutAction();
		WareHouse.M_ResetFeedInBox();
		WareHouse.M_ResetReloadBox();
		uiResettingStep := 100;
	100:
		_ResetCompleted := TRUE;
END_CASE
IF _ResetCompleted THEN
    eState := STATE_DORMANT;
END_IF
END_METHOD

END_FUNCTION_BLOCK

// ---- Library/20_MachineUnits/21_StorageArea/210_Cabinet/FB_WareHouse.TcPOU
FUNCTION_BLOCK FB_WareHouse EXTENDS FB_Objectbase
VAR_INPUT
	 Motors 		  : REFERENCE TO UNI_MotorList;
	 WheelhouseSensor : REFERENCE TO UNI_HMI_WheelHouseInput;
END_VAR
VAR_OUTPUT
END_VAR
VAR
   
    nMotorIndex    : UINT;
    CabinetJob     : E_CabinetJob := E_CabinetJob.Idle;    

    stLayerStatus    : st_LayerStatus;
    stWarehouseLayer : st_WarehouseLayer;
    stWarehouseList  : st_WarehouseList;
    _stWarehouseList : _st_WarehouseList;

	fbReloadBox : FB_ReloadBox;
	fbFeedInBox : FB_FeedInBox;
END_VAR

SUPER^.M_clcUpdate();
THIS^.M_clcUpdate();

PROPERTY PUBLIC bFeedInBox_Completed : BOOL
GET
bFeedInBox_Completed := fbFeedInBox.Done;
END_GET
END_PROPERTY

PROPERTY bReloadBox_Completed : BOOL
GET
bReloadBox_Completed := fbReloadBox.Done;
END_GET
END_PROPERTY

METHOD M_clcFBs : BOOL
VAR_INPUT	
END_VAR
VAR
	nELIndex			:	INT;
END_VAR
fbReloadBox(
	Execute:= , 
	Abort:= , 
	Reset:= , 
	ObjectName:= 'Warehouse Reload box', 
	Busy=> bBusy, 
	Done=> bDone, 
	Aborted=> , 
	Error=> bError, 
	ErrorID=> , 
	Status=> , 
	Motors:= Motors, 
	WarehouseStatus:= WheelhouseSensor.List, 
	ArrivedDelayTime:= T#1S, 
	WarehouseSelect:= , 
	WarehouseCoordinates:= , 
	TimeOut:= T#10S);
	
fbFeedInBox(
	Execute:= , 
	Abort:= , 
	Reset:= , 
	ObjectName:= 'Warehouse FeedIn box', 
	Busy=> bBusy, 
	Done=> bDone, 
	Aborted=> , 
	Error=> bError, 
	ErrorID=> , 
	Status=> , 
	Motors:= Motors, 
	WarehouseStatus:= WheelhouseSensor.List, 
	ArrivedDelayTime:= T#2.0S, 
	WarehouseSelect:= , 
	WarehouseCoordinates:= , 
	TimeOut:= T#10S);
END_METHOD

METHOD M_clcUpdate : BOOL
VAR_INPUT	
END_VAR
VAR	
	i : INT;
END_VAR
//clc FBs
M_clcFBs();
END_METHOD

METHOD PRIVATE M_GotoCommandStep : BOOL
VAR_INPUT
END_VAR
CabinetJob := E_CabinetJob.Initial;
END_METHOD

METHOD PRIVATE M_GotoErrorStep : BOOL
VAR_INPUT
END_VAR
CabinetJob := E_CabinetJob.error;
END_METHOD

METHOD PUBLIC M_ResetFeedInBox : BOOL
VAR_INPUT
END_VAR
VAR
	uiMotorInder : UINT; 
END_VAR
// reset reload box execute
fbFeedInBox.Execute := FALSE;
 
M_ResetFeedInBox := TRUE; // Method end
END_METHOD

METHOD M_ResetReloadBox : Bool
VAR_INPUT
END_VAR
// reset reload box execute
fbReloadBox.Execute := FALSE;

M_ResetReloadBox := true; // Method end
END_METHOD

METHOD PUBLIC M_StartFeedInBox : BOOL
VAR_INPUT
	WareHouseSelect : E_WareHouse;
	WarehouseCoordinates : ST_WareHouseCoordinates;
END_VAR
// Send command to Feedin box fb
fbFeedInBox.WarehouseSelect := WareHouseSelect;
fbFeedInBox.WarehouseCoordinates := WarehouseCoordinates;
fbFeedInBox.Execute := TRUE;

M_StartFeedInBox := TRUE; // Method end
END_METHOD

METHOD M_StartReloadBox : BOOL
VAR_INPUT
	WareHouseSelect : E_WareHouse;
	WarehouseCoordinates : ST_WareHouseCoordinates;
END_VAR
// Send command to reload box fb
fbReloadBox.WarehouseSelect := WareHouseSelect;
fbReloadBox.WarehouseCoordinates := WarehouseCoordinates;
fbReloadBox.Execute := TRUE;

M_StartReloadBox := true; // Method end
END_METHOD

END_FUNCTION_BLOCK

// ---- POUs/ModbusRTU/00_BaseFBs/01_FB_ObjectBase/FB_ObjectBase.TcPOU
FUNCTION_BLOCK FB_ObjectBase

VAR
	{attribute 'hide'}
	fbLocalSystemTime				: FB_LocalSystemTime := (bEnable := TRUE, dwCycle := 1);
	{attribute 'hide'}
	uiCmdIndex						: UINT := 1;
	arCmdRecord						: ARRAY[1..Para_ObjectBase.cNumCmdRecord] OF ST_CmdContent;
	{attribute 'hide'}
	uiMsgIndex						: UINT := 1;
	arMsgRecord						: ARRAY[1..Para_ObjectBase.cNumMsgRecord] OF ST_MsgContent;
	{attribute 'hide'}
	bReset							: BOOL;
END_VAR

VAR_OUTPUT
	bBusy							: BOOL;
	bDone							: BOOL;
	bError							: BOOL;
	sErrMessage						: STRING;
END_VAR

(* Info - Please update if you modify something. =========================
Create Date	: 2023/12/12
Last Update	: 2023/12/15
Description	: Base object for "Unit" FB to extend.
			  Provide basic status method and record function.
			  Please extend this FB and call super^() in your FB.
Change Log	: 2023/12/12 -> Add Reset method, user should clear after reseting done.
			  2023/12/13 -> Debug ErrMessage logic.
			  2023/12/15 -> Add command record when reseting.
=========================================================================*)

THIS^.M_clcUpdate();

METHOD  M_clcUpdate : BOOL
VAR_INPUT
END_VAR
fbLocalSystemTime();
IF bError THEN
	IF uiMsgIndex > 1 THEN
		sErrMessage := arMsgRecord[uiMsgIndex-1].Message;
	END_IF
ELSE
	sErrMessage := '';
END_IF
END_METHOD

METHOD M_RecordCmd : BOOL
VAR_INPUT
	sSource					: STRING;
	sCommand				: STRING;
END_VAR
arCmdRecord[uiCmdIndex].SysTime := SYSTEMTIME_TO_STRING(fbLocalSystemTime.systemTime);
arCmdRecord[uiCmdIndex].Source := sSource;
arCmdRecord[uiCmdIndex].Command := sCommand;

uiCmdIndex := uiCmdIndex + 1;
IF uiCmdIndex > Para_ObjectBase.cNumCmdRecord THEN uiCmdIndex := 1; END_IF

M_RecordCmd := TRUE;
END_METHOD

METHOD M_RecordMsg : BOOL
VAR_INPUT
	sSource					: STRING;
	sMessgae				: STRING;
END_VAR
arMsgRecord[uiMsgIndex].SysTime := SYSTEMTIME_TO_STRING(fbLocalSystemTime.systemTime);
arMsgRecord[uiMsgIndex].Source := sSource;
arMsgRecord[uiMsgIndex].Message := sMessgae;

uiMsgIndex := uiMsgIndex + 1;
IF uiMsgIndex > Para_ObjectBase.cNumMsgRecord THEN uiMsgIndex := 1; END_IF

M_RecordMsg := TRUE;
END_METHOD

METHOD M_Reset : BOOL
VAR_INPUT
    sRecordSource :STRING;
END_VAR
IF bError THEN
	bReset := TRUE;
	M_RecordCmd(sSource:=sRecordSource, sCommand:='Reset');
END_IF
END_METHOD

METHOD M_SearchCommand : ST_CmdContent
VAR_INPUT
	uiCmdIndex				: UINT;
END_VAR
IF uiCmdIndex > 0 AND uiCmdIndex <= Para_ObjectBase.cNumCmdRecord THEN
	M_SearchCommand := arCmdRecord[uiCmdIndex];
END_IF
END_METHOD

METHOD M_SearchMessage : ST_MsgContent
VAR_INPUT
	uiMsgIndex				: UINT;
END_VAR
IF uiMsgIndex > 0 AND uiMsgIndex <= Para_ObjectBase.cNumMsgRecord THEN
	M_SearchMessage := arMsgRecord[uiMsgIndex];
END_IF
END_METHOD

METHOD M_SetBusy : BOOL
VAR_INPUT
END_VAR
THIS^.bBusy := TRUE;
THIS^.bDone := FALSE;
THIS^.bError := FALSE;
END_METHOD

METHOD M_SetDone : BOOL
VAR_INPUT
END_VAR
THIS^.bBusy := FALSE;
THIS^.bDone := TRUE;
THIS^.bError := FALSE;
END_METHOD

METHOD M_SetError : BOOL
VAR_INPUT
END_VAR
THIS^.bBusy := FALSE;
THIS^.bDone := FALSE;
THIS^.bError := TRUE;
END_METHOD

PROPERTY P_Busy : BOOL
GET
P_Busy := THIS^.bBusy;
END_GET
END_PROPERTY

PROPERTY P_Done : BOOL
GET
P_Done := THIS^.bDone;
END_GET
END_PROPERTY

{attribute 'monitoring' := 'variable'}
PROPERTY P_Error : BOOL
GET
P_Error := THIS^.bError;
END_GET
END_PROPERTY

PROPERTY P_ErrorMessage : STRING
GET
P_ErrorMessage := THIS^.sErrMessage;
END_GET
END_PROPERTY

END_FUNCTION_BLOCK

// ---- Library/20_MachineUnits/21_StorageArea/210_Cabinet/Services/FB_ReloadBox.TcPOU
FUNCTION_BLOCK FB_ReloadBox EXTENDS FB_ObjectBase_V2 IMPLEMENTS IBasicElement
VAR_INPUT
	Motors : REFERENCE TO UNI_MotorList ;// The motors with warehouse conveyor
	WarehouseStatus : REFERENCE TO ST_WheelhouseInput; // The warehouse motor and sensor status
	ArrivedDelayTime : TIME;
	WarehouseSelect :E_WareHouse;
	WarehouseCoordinates : ST_WareHouseCoordinates;
	TimeOut : TIME; // Set the time if the process stop
END_VAR
VAR_OUTPUT
END_VAR
VAR
	Ton_ArriveDelay : TON; // When box arrived the front sensor, delay some time.
	Ton_BoxMoveForward : TON;// When the conveyor send the box forward, but not useful.
	uiMotorIndex: INT;
	CurrentTargetSensorStatus : BOOL;
END_VAR

A00_BasicUnits();
A10_StateControl();

ACTION A00_BasicUnits:
// Timer
Ton_ArriveDelay(PT:= ArrivedDelayTime);
Ton_BoxMoveForward(PT:= TimeOut);
END_ACTION

(* Check Warehouse front sensor status
*)
METHOD M_CheckSlideSensor
VAR_INPUT
    WarehouseSelect      : E_WareHouse;
    WarehouseCoordinates : ST_WareHouseCoordinates;
END_VAR
VAR_OUTPUT
	SensorStatus : BOOL;
END_VAR
IF WarehouseSelect = E_WareHouse.WareHouseA THEN
    SensorStatus := WarehouseStatus.WheelhouseA.arLayer[WarehouseCoordinates.Layer].Line[WarehouseCoordinates.Slide];
ELSIF WarehouseSelect = E_WareHouse.WareHouseB THEN
    SensorStatus := WarehouseStatus.WheelhouseB.arLayer[WarehouseCoordinates.Layer].Line[WarehouseCoordinates.Slide];
END_IF
END_METHOD

METHOD  M_STATE_ABORTED
VAR_INPUT
END_VAR
END_METHOD

METHOD  M_STATE_ABORTING
VAR_INPUT
END_VAR
END_METHOD

METHOD  M_STATE_DONE
VAR_INPUT
END_VAR
Busy := FALSE;
Done := _Executed;
IF NOT Execute THEN
	eState := STATE_RESETTING;
END_IF
END_METHOD

METHOD  M_STATE_DORMANT
VAR_INPUT
END_VAR
// Clear FB output
Busy            := FALSE;
Done            := FALSE;
Aborted         := FALSE;
Error           := FALSE;
ErrorID         := 0;
Status          := '';
_ResetCompleted := FALSE;
_Error          := FALSE;
_Executed       := FALSE;
Ton_ArriveDelay.IN := FALSE;
Ton_BoxMoveForward.IN := FALSE;
uiExecutingStep := 0;
CurrentTargetSensorStatus := FALSE;
// Wait Execute command
IF Execute THEN
    eState := STATE_EXECUTING;
END_IF
END_METHOD

METHOD  M_STATE_ERROR
VAR_INPUT
END_VAR
FOR uiMotorIndex := 1 TO 20 DO
	Motors.arMotor[uiMotorIndex].M_MotorStop();// 
END_FOR

IF NOT Execute THEN
	estate := STATE_RESETTING;
END_IF
END_METHOD

METHOD  M_STATE_EXECUTING
VAR_INPUT
END_VAR
VAR_INST
	TargetLayer : INT;
	TargetSlide :E_WareHouseSlide;
END_VAR
// Set FB state is busy
Busy := TRUE;

// Process
CASE uiExecutingStep OF
    0: // Command analize
		 Ton_ArriveDelay.IN := FALSE;
		 TargetLayer := WarehouseCoordinates.Layer+(WarehouseSelect-1)*10; //Warehouse A = 1 , B = 2
		 TargetSlide := WarehouseCoordinates.Slide;
		uiExecutingStep := 10;
	10:
		 Ton_BoxMoveForward.IN := TRUE;
        Motors.arMotor[TargetLayer].M_MoveForward();// .M_MoveForward();//('Reload box : conveyor move forward');
		IF NOT Motors.arMotor[TargetLayer].InStopped THEN// .InStopped;// THEN
			Ton_BoxMoveForward.IN := FALSE;
			uiExecutingStep := 100;
		END_IF
		IF  Ton_BoxMoveForward.Q THEN
		  _Error := TRUE;
           Status := 'Move motor timeout';
		END_IF
    100: // Wait box arrived
        Ton_BoxMoveForward.IN := TRUE;
		M_CheckSlideSensor(WarehouseSelect := WarehouseSelect, WarehouseCoordinates := WarehouseCoordinates,SensorStatus=>CurrentTargetSensorStatus);
        Ton_ArriveDelay.IN:=CurrentTargetSensorStatus;

		IF Ton_ArriveDelay.Q THEN
            uiExecutingStep := 200;
//        ELSIF Ton_BoxMoveForward.Q THEN
//            _Error := TRUE;
//            Status := 'Box was not been arrived,time out';
        END_IF
    200:
        Ton_ArriveDelay.IN := FALSE;

        //IF Ton_ArriveDelay.Q THEN
            uiExecutingStep := 300;
       // END_IF
    300:
        Motors.arMotor[TargetLayer].M_MotorStop();// .M_MotorStop();//('Reload box : conveyor move forward');
        uiExecutingStep := 9900;
    9900:
        // Command completed
        _Executed := TRUE;
END_CASE

IF _Executed THEN
    eState := STATE_DONE;
ELSIF NOT Execute THEN
    eState := STATE_RESETTING;
ELSIF _Error THEN
    eState := STATE_ERROR;
END_IF
END_METHOD

METHOD  M_STATE_RESETTING
VAR_INPUT
END_VAR
VAR 
	uiMotorIndex : UINT;
END_VAR
Done := _Executed;
		Ton_BoxMoveForward.IN := FALSE;
		Ton_ArriveDelay.IN := FALSE;
FOR uiMotorIndex := 1 TO 20 DO 
	Motors.arMotor[uiMotorIndex].M_MotorStop();
END_FOR		
		
IF NOT Execute THEN
	eState := STATE_DORMANT;
END_IF
END_METHOD

END_FUNCTION_BLOCK

// ---- Library/20_MachineUnits/21_StorageArea/210_Cabinet/Services/FB_FeedInBox.TcPOU
FUNCTION_BLOCK FB_FeedInBox EXTENDS FB_ObjectBase_V2 IMPLEMENTS IBasicElement
VAR_INPUT
	Motors : REFERENCE TO UNI_MotorList ; // The motors with warehouse conveyor
	WarehouseStatus : REFERENCE TO ST_WheelhouseInput; // The warehouse motor and sensor status
	ArrivedDelayTime : TIME;
	WarehouseSelect :E_WareHouse;
	WarehouseCoordinates : ST_WareHouseCoordinates;
	TimeOut : TIME; // Set the time if the process stop
END_VAR
VAR_OUTPUT
END_VAR
VAR
	Ton_ArriveDelay : TON; // When box arrived the front sensor, delay some time.
	Ton_BoxMoveForward : TON;// When the conveyor send the box forward, but not useful.
	tonFirstReserveTime	:TON;
	tonSecondForwardTime	:TON;
	tonThirdReserceTime	:TON;
	uiMotorIndex: INT;
	CurrentTargetSensorStatus : BOOL;
END_VAR

A00_BasicUnits();
A10_StateControl();

ACTION A00_BasicUnits:
// Timer
Ton_ArriveDelay(PT:= ArrivedDelayTime);//2.0s
Ton_BoxMoveForward(PT:= TimeOut);//10S

//check full box in cabinet time
tonFirstReserveTime(PT :=T#1.5S);	
tonSecondForwardTime(PT :=T#750MS);
tonThirdReserceTime(PT :=T#2.0S);
END_ACTION

(* Check Warehouse front sensor status
*)
METHOD M_CheckSlideSensor
VAR_INPUT
    WarehouseSelect      : E_WareHouse;
    WarehouseCoordinates : ST_WareHouseCoordinates;
END_VAR
VAR_OUTPUT
	SensorStatus : BOOL;
END_VAR
IF WarehouseSelect = E_WareHouse.WareHouseA THEN
    SensorStatus := WarehouseStatus.WheelhouseA.arLayer[WarehouseCoordinates.Layer].Line[WarehouseCoordinates.Slide];
ELSIF WarehouseSelect = E_WareHouse.WareHouseB THEN
    SensorStatus := WarehouseStatus.WheelhouseB.arLayer[WarehouseCoordinates.Layer].Line[WarehouseCoordinates.Slide];
END_IF
END_METHOD

METHOD  M_STATE_ABORTED
VAR_INPUT
END_VAR
END_METHOD

METHOD  M_STATE_ABORTING
VAR_INPUT
END_VAR
END_METHOD

METHOD  M_STATE_DONE
VAR_INPUT
END_VAR
Busy := FALSE;
Done := TRUE;
IF NOT Execute THEN
	eState := STATE_RESETTING;
END_IF
END_METHOD

METHOD  M_STATE_DORMANT
VAR_INPUT
END_VAR
// Clear FB output
Busy            := FALSE;
Done            := FALSE;
Aborted         := FALSE;
Error           := FALSE;
ErrorID         := 0;
Status          := '';
_ResetCompleted := FALSE;
_Error          := FALSE;
_Executed       := FALSE;
Ton_ArriveDelay.IN := FALSE;
Ton_BoxMoveForward.IN := FALSE;
tonFirstReserveTime.IN :=FALSE;
tonSecondForwardTime.IN :=FALSE;
tonThirdReserceTime.IN :=FALSE;
uiExecutingStep := 0;
CurrentTargetSensorStatus := FALSE;
// Wait Execute command
IF Execute THEN
    eState := STATE_EXECUTING;
END_IF
END_METHOD

METHOD  M_STATE_ERROR
VAR_INPUT
END_VAR
FOR uiMotorIndex := 1 TO 20 DO
	Motors.arMotor[uiMotorIndex].M_MotorStop();
END_FOR

IF NOT Execute THEN
	estate := STATE_RESETTING;
END_IF
END_METHOD

